// When zones get deleted on tracking end, the remaining distance to move reserved zones
// is limited to the windows up to the absolute window positions and the trackinglength backwards.
// Therefore from all windows of a TrackingLength - Startwindow is the distance 
// to be removed from the allowed shifting distance.
StartTrackingPosition := M_GetTrackingPosition((mStartWindowIndex-1)*WindowSize);
WindowsFromBegin := UDINT_TO_UINT(StartTrackingPosition / WindowSize);
WindowsTrackingLength := UDINT_TO_UINT((TrackingLength + TrackingAddition) / WindowSize);

IF WindowsFromBegin MOD WindowSize > 0 THEN
	WindowsFromBegin := WindowsFromBegin + 1;
END_IF

IF WindowsTrackingLength MOD WindowSize > 0 THEN
	WindowsTrackingLength := WindowsTrackingLength + 1;
END_IF

IF DeleteZoneTrackingEnd THEN	
	RemainingWindowLength := UINT_TO_INT(WindowsFromBegin) + UINT_TO_INT(WindowsTrackingLength) - UINT_TO_INT(ResWindowsToShift) - 1;
ELSE
	RemainingWindowLength := UINT_TO_INT(MaxWindowIndex) - UINT_TO_INT(ResWindowsToShift) - 1;
END_IF
	
FOR mIdx := 1 TO WindowTracking.MAX_NUMBER_OF_WINDOWS DO
	// Correct window border overflow
	IF mWindowIndex > MaxWindowIndex THEN
		mWindowIndex := mWindowIndex - MaxWindowIndex;
	END_IF
	
	IF mNextTargetWindow > MaxWindowIndex THEN
		mNextTargetWindow := mNextTargetWindow - MaxWindowIndex;
	END_IF
	
	// Relocation is done, if all zones in the shifting distance
	// and all interfering zones are relocated properly
	IF mIdx > ResWindowsToShift THEN
		M_IsShiftable := TRUE;
		EXIT;

	// If window is part of zone, try to schedule relocation
	ELSIF WindowTable[mWindowIndex].ZoneIndex > 0 THEN
		// Calculate Window Length of Zone which should be relocated
		mZoneIndexReloc := WindowTable[mWindowIndex].ZoneIndex;
		
		IF ZoneTable[mZoneIndexReloc].TU_Present THEN
			// Skip all occupied zones, because they are not allowed for re-allocation, otherwise fail
			IF mExcludeTUs THEN
				mWindowIndex := mWindowIndex + 1;
				RemainingWindowLength := RemainingWindowLength - 1;
				CONTINUE;
			ELSE
				M_IsShiftable := FALSE;
				EXIT;
			END_IF
		END_IF

		IF ZoneTable[mZoneIndexReloc].ZoneEndWindowIndex > ZoneTable[mZoneIndexReloc].ZoneStartWindowIndex THEN
			mWindowLength := ZoneTable[mZoneIndexReloc].ZoneEndWindowIndex - ZoneTable[mZoneIndexReloc].ZoneStartWindowIndex + 1;
		ELSE
			mWindowLength := ZoneTable[mZoneIndexReloc].ZoneEndWindowIndex + MaxWindowIndex  - ZoneTable[mZoneIndexReloc].ZoneStartWindowIndex + 1;
		END_IF

		// Check if reallocation would overwrite start point
		IF RemainingWindowLength - UINT_TO_INT(mWindowLength) > 0 THEN
			RelocScheduled := mfbRelocator.M_ScheduleRelocation(
									mZoneIndex				:= mZoneIndexReloc, 
									mTargetWindow			:= mNextTargetWindow, 
									mMaxWindowIndex			:= MaxWindowIndex, 
									mrWindowTable			:= WindowTable, 
									mrZoneTable				:= ZoneTable, 
									mBlockingZoneIndex		=> BlockingZoneIndex, 
									mBlockingEndWindowIndex => BlockingEndWindowIndex,
									mErrorId				=> ErrorId);
									
			// If relocation could be scheduled properly
			// set next window to the window after the relocated zone
			IF RelocScheduled THEN
				mNextTargetWindow := mNextTargetWindow + mWindowLength;
				
				// Adjust index of next window to check if relocation was successful
				mWindowIndex := mWindowIndex + mWindowLength;
				
				// Each found zone on the shifting distance requires one additional shift iteration
				// Because the location where it was moved to, may contains as well a zone which needs to be shifted
				ResWindowsToShift := ResWindowsToShift + 1;
				
				// Ensure that reallocation does not overwrite start point
				RemainingWindowLength := RemainingWindowLength - UINT_TO_INT(mWindowLength);
			ELSE
				// Relocation was not possible because of a Zone which is not allowed
				// to be shifted, try again with window after the blocking zone
				IF BlockingZoneIndex > 0 THEN
					// Each found zone on the shifting distance requires one additional shift iteration
					ResWindowsToShift := ResWindowsToShift + 1;
					
					// Calc length of blocking zone
					IF ZoneTable[BlockingZoneIndex].ZoneEndWindowIndex >= ZoneTable[BlockingZoneIndex].ZoneStartWindowIndex THEN
						mWindowLengthBlocking := ZoneTable[BlockingZoneIndex].ZoneEndWindowIndex - ZoneTable[BlockingZoneIndex].ZoneStartWindowIndex;
					ELSE
						mWindowLengthBlocking := ZoneTable[BlockingZoneIndex].ZoneEndWindowIndex + MaxWindowIndex - ZoneTable[BlockingZoneIndex].ZoneStartWindowIndex;
					END_IF
					
					mNextTargetWindow := BlockingEndWindowIndex + 1;
					
					RemainingWindowLength := RemainingWindowLength - UINT_TO_INT(mWindowLengthBlocking);
				END_IF
			END_IF
		ELSE
			// The found zone could not be placed on the tracking because there is no space left.
			// Mark overrun and leave
			mZoneOverrun := TRUE;
			mZoneOverrunWindowIndex := mWindowIndex;
			M_IsShiftable := mAllowOverrun;
			EXIT;
		END_IF
	ELSE
		mWindowIndex := mWindowIndex + 1;
		RemainingWindowLength := RemainingWindowLength - 1;
	END_IF
END_FOR
END_METHOD

/// Checks if a TU or a part of it, is found in a certain range.
METHOD M_IsTU_InRange : BOOL; // Returns true if present, otherwise false
VAR_INPUT
	mZoneIndex				: UINT; // Tracking zone index
	mAbsoluteStartRange		: UDINT; // Start range position on the tracking [mm]
	mAbsoluteEndRange		: UDINT; // End range position on the tracking [mm]
END_VAR
VAR
	mStartWindowIndex		: UINT; // Window index at start position
	mEndWindowIndex			: UINT; // Window index at end position
	mTrackingRangeEnd		: UDINT; // Tracking range position end
	mTrackingRangeStart		: UDINT; // Tracking range position start
	mTrackingTU_End			: UDINT; // Tracking range position end
	mTrackingTU_Start		: UDINT; // Tracking range position start
END_VAR
M_IsTU_InRange := FALSE;

// Check inputs
IF mZoneIndex = 0 THEN
	RETURN;
END_IF

IF NOT ZoneTable[mZoneIndex].TU_Present THEN
	RETURN;
END_IF

// Get window index of window start position
mStartWindowIndex := M_GetWindowIndex(mAbsoluteStartRange);
// Get window index of window end position
mEndWindowIndex := M_GetWindowIndex(mAbsoluteEndRange);

// Remark:
// Absolute view is unequal to tracking view
// ABS:  500mm 505mm .....1000mm
//   AbsStartpos		AbsEndPos
//       |                  |
//    TrackingEnd       TrackingStart
//
//  --------------------------------------      FlowDirection ->
// Win:  54  53  52 ....  43 42 ...
// Window index of end is normally lower than start (except overflow)     

// Ensure both window index are in a valid range
IF mStartWindowIndex > 0 AND mStartWindowIndex <= WindowTracking.MAX_NUMBER_OF_WINDOWS AND
   mEndWindowIndex > 0 AND mEndWindowIndex <= WindowTracking.MAX_NUMBER_OF_WINDOWS THEN
	
	// Ensure that Zone consists of start and end tu window index
	IF ZoneTable[mZoneIndex].TU_StartWindowIndex > 0 AND
	   ZoneTable[mZoneIndex].TU_EndWindowIndex > 0 THEN
	   
		//    TrackingEnd       TrackingStart
		//         |-----------------|
		//  --------------------------------------      FlowDirection ->
	   	mTrackingTU_End := WindowTable[ZoneTable[mZoneIndex].TU_EndWindowIndex].TU_RearEdgePosition;
	   	mTrackingTU_Start :=  WindowTable[ZoneTable[mZoneIndex].TU_StartWindowIndex].TU_FrontEdgePosition;
	   
		//    TrackingRangeEnd  TrackingRangeStart
		//      |----------------------|
		//  --------------------------------------      FlowDirection ->
		mTrackingRangeEnd := M_GetTrackingPosition(mAbsoluteStartRange);
   		mTrackingRangeStart := M_GetTrackingPosition(mAbsoluteEndRange);
	   
		// When range does not consists of the overflow point
		IF mTrackingRangeEnd >= mTrackingRangeStart THEN 
			// Check if TU End edge is between range
			IF mTrackingTU_End >= mTrackingRangeStart AND
               mTrackingTU_End <= mTrackingRangeEnd THEN
				M_IsTU_InRange := TRUE;
				RETURN;
				
			// Check if TU start edge is between range
			ELSIF mTrackingTU_Start >= mTrackingRangeStart AND
                  mTrackingTU_Start <= mTrackingRangeEnd THEN
				M_IsTU_InRange := TRUE;
				RETURN;
				
			// Check if TU is overlapping full range
			ELSIF mTrackingTU_End >= mTrackingRangeEnd AND
                  mTrackingTU_Start <= mTrackingRangeStart THEN
				M_IsTU_InRange := TRUE;
				RETURN; 
			END_IF
		// If range is overlapping overflow point
		ELSE
			// Check if TU End edge is between range
			IF mTrackingTU_End >= mTrackingRangeStart OR  
               mTrackingTU_End <= mTrackingRangeEnd THEN
				M_IsTU_InRange := TRUE;
				RETURN;
				
			// Check if TU start edge is between range
			ELSIF mTrackingTU_Start >= mTrackingRangeStart OR  
               mTrackingTU_Start <= mTrackingRangeEnd THEN
				M_IsTU_InRange := TRUE;
				RETURN;
				
			// Check if TU is overlapping full range
			ELSIF mTrackingTU_End >= mTrackingRangeEnd AND
                  mTrackingTU_Start <= mTrackingRangeStart THEN
				M_IsTU_InRange := TRUE;
				RETURN; 
			END_IF
		END_IF
	END_IF
END_IF
END_METHOD

/// Returns if a physical TU is present at mAbsolutePosition
METHOD M_IsTU_Present : BOOL; // Returns true if present, otherwise false
VAR_INPUT
	mAbsolutePosition		: UDINT; // Absolute position on tracking length
END_VAR
VAR
	mWindowIndex			: UINT; // Window index at absolute position
	mTrackingPosition		: UDINT; // Current position on tracking
END_VAR
M_IsTU_Present := FALSE;

// Get window index of position
mWindowIndex := M_GetWindowIndex(mAbsolutePosition);

IF mWindowIndex > 0 AND mWindowIndex <= WindowTracking.MAX_NUMBER_OF_WINDOWS THEN
	// Get position on tracking
	mTrackingPosition := M_GetTrackingPosition(mAbsolutePosition);

	// Get TU state
	CASE WindowTable[mWindowIndex].State OF
		E_WindowTrackingWindowState.IDLE:
			M_IsTU_Present := FALSE;
			
		E_WindowTrackingWindowState.FRONT_EDGE:
			IF WindowTable[mWindowIndex].TU_FrontEdgePosition <= mTrackingPosition THEN
				M_IsTU_Present := TRUE;
			ELSE
				M_IsTU_Present := FALSE;
			END_IF
		
		E_WindowTrackingWindowState.REAR_EDGE:
			IF WindowTable[mWindowIndex].TU_RearEdgePosition > mTrackingPosition THEN
				M_IsTU_Present := TRUE;
			ELSE
				M_IsTU_Present := FALSE;
			END_IF
		
		E_WindowTrackingWindowState.OCCUPIED:
			M_IsTU_Present := TRUE;
	END_CASE
END_IF
END_METHOD

/// Checks if a zone or a part of it,  is found in a certain range.
METHOD M_IsZoneInRange : BOOL; // Returns true if zone is in range, otherwise false
VAR_INPUT
	mZoneIndex				: UINT; // Tracking zone index
	mAbsoluteStartRange		: UDINT; // Start range position on the tracking [mm]
	mAbsoluteEndRange		: UDINT; // End range position on the tracking [mm]
END_VAR
VAR
	mStartWindowIndex		: UINT; // Window index at start position
	mEndWindowIndex			: UINT; // Window index at end position
	mTrackingRangeEnd		: UDINT; // Tracking range position end
	mTrackingRangeStart		: UDINT; // Tracking range position start
	mTrackingZoneEnd		: UDINT; // Tracking range position zone end
	mTrackingZoneStart		: UDINT; // Tracking range position zone start
END_VAR
M_IsZoneInRange := FALSE;

// Check inputs
IF mZoneIndex = 0 THEN
	RETURN;
END_IF

// Get window index of window start position
mStartWindowIndex := M_GetWindowIndex(mAbsoluteStartRange);
// Get window index of window end position
mEndWindowIndex := M_GetWindowIndex(mAbsoluteEndRange);

// Remark:
// Absolute view is unequal to tracking view
// ABS:  500mm 505mm .....1000mm
//    Startpos			 EndPos
//       |                  |
//  --------------------------------------      FlowDirection ->
// Win:  54  53  52 ....  43 42 ...
// Window index of end is normally lower than start (except overflow)     

// Ensure both window index are in a valid range
IF mStartWindowIndex > 0 AND mStartWindowIndex <= WindowTracking.MAX_NUMBER_OF_WINDOWS AND
   mEndWindowIndex > 0 AND mEndWindowIndex <= WindowTracking.MAX_NUMBER_OF_WINDOWS THEN

	// Ensure that Zone consists of start and end tu window index
	IF ZoneTable[mZoneIndex].TU_StartWindowIndex > 0 AND
	   ZoneTable[mZoneIndex].TU_EndWindowIndex > 0 THEN

		//    TrackingEnd       TrackingStart
		//         |-----------------|
		//  --------------------------------------      FlowDirection ->
	   	mTrackingZoneEnd := ZoneTable[mZoneIndex].ZoneEndPosition;
	   	mTrackingZoneStart := ZoneTable[mZoneIndex].ZoneStartPosition;

		//    TrackingRangeEnd  TrackingRangeStart
		//      |----------------------|
		//  --------------------------------------      FlowDirection ->
		mTrackingRangeEnd := M_GetTrackingPosition(mAbsoluteStartRange);
   		mTrackingRangeStart := M_GetTrackingPosition(mAbsoluteEndRange);

		// When range does not consists of the overflow point
		IF mTrackingRangeEnd >= mTrackingRangeStart THEN 
			// Check if TU End edge is between range
			IF mTrackingZoneEnd >= mTrackingRangeStart AND
               mTrackingZoneEnd <= mTrackingRangeEnd THEN
				M_IsZoneInRange := TRUE;
				RETURN;
				
			// Check if TU start edge is between range
			ELSIF mTrackingZoneStart >= mTrackingRangeStart AND
                  mTrackingZoneStart <= mTrackingRangeEnd THEN
				M_IsZoneInRange := TRUE;
				RETURN;
				
			// Check if TU is overlapping full range
			ELSIF mTrackingZoneEnd >= mTrackingRangeEnd AND
                  mTrackingZoneStart <= mTrackingRangeStart THEN
				M_IsZoneInRange := TRUE;
				RETURN; 
			END_IF
			
		// If range is overlapping overflow point
		ELSE
			// Check if TU End edge is between range
			IF mTrackingZoneEnd >= mTrackingRangeStart OR  
               mTrackingZoneEnd <= mTrackingRangeEnd THEN
				M_IsZoneInRange := TRUE;
				RETURN;
				
			// Check if TU start edge is between range
			ELSIF mTrackingZoneStart >= mTrackingRangeStart OR  
                  mTrackingZoneStart <= mTrackingRangeEnd THEN
				M_IsZoneInRange := TRUE;
				RETURN;
				
			// Check if TU is overlapping full range
			ELSIF mTrackingZoneEnd >= mTrackingRangeEnd AND
                  mTrackingZoneStart <= mTrackingRangeStart THEN
				M_IsZoneInRange := TRUE;
				RETURN; 
			END_IF
		END_IF
	END_IF
END_IF
END_METHOD

/// Tries to free a certain area by the following options (Shift, Shorten, Delete)
METHOD PROTECTED M_MakeSpace : BOOL // Returns true if successfully
VAR_INPUT
	mStartWindowIndex		: UINT; // Start window index
	mWindowsToFree			: UINT; // Windows to free up (e.g. 1 only clears start window index)
	mAllowZoneDelete		: BOOL; // Allows to delete zones if they could not be modified or reloacted
END_VAR
VAR_INST
	MinFreeWindowIndex		: UINT; // Minimum window index until space has to be free 
	ShiftZonesOk			: BOOL; // Shift was executed
END_VAR
VAR
	mIdx					: UINT; // Iteration
	mWindowIndex			: UINT; // Temp window index
	mZoneIndex				: UINT; // Zone index
	mTU_StartInArea			: BOOL; // TU start found in area
	mTU_EndInArea			: BOOL; // TU end found in area
END_VAR
// Initialize
M_MakeSpace := FALSE;

// Validate inputs
IF mStartWindowIndex = 0 OR
   mStartWindowIndex > WindowTracking.MAX_NUMBER_OF_WINDOWS OR
   mWindowsToFree = 0 OR
   mWindowsToFree > WindowTracking.MAX_NUMBER_OF_WINDOWS OR
   WindowSize = 0 THEN
	RETURN;
END_IF

// Initialize for-loop values
mWindowIndex := mStartWindowIndex;

// Calculate minimum window index which has to be free 
// Example: Startwindow 49, windows to be free 4 (49, 50, 51, 52)
//                  |-------------->
// Window     53 | 52 | 51 | 50 | 49
MinFreeWindowIndex := mStartWindowIndex + mWindowsToFree - 1;
	
// Correct window border overflow
IF MinFreeWindowIndex > MaxWindowIndex THEN
	MinFreeWindowIndex := MinFreeWindowIndex - MaxWindowIndex;
END_IF

// Check for any occupied zone in the area to be free and test if it spossible to shorten or delete it
FOR mIdx := 1 TO mWindowsToFree DO	
	IF WindowTable[mWindowIndex].ZoneIndex > 0 THEN
		mZoneIndex := WindowTable[mWindowIndex].ZoneIndex;
	
		// Zone can be modified by one of the following options
		// - If Occupied -> Shorten
		// - Else Delete if allowed
		IF ZoneTable[mZoneIndex].TU_Present THEN
			// Shorten
			// Check if position of TU inside the zone is outside of the area to be free
			IF MinFreeWindowIndex >= mStartWindowIndex THEN
				mTU_StartInArea := ZoneTable[mZoneIndex].TU_StartWindowIndex >= mStartWindowIndex AND
				   				   ZoneTable[mZoneIndex].TU_StartWindowIndex <= MinFreeWindowIndex;
				
				mTU_EndInArea := ZoneTable[mZoneIndex].TU_EndWindowIndex >= mStartWindowIndex AND
				   				 ZoneTable[mZoneIndex].TU_EndWindowIndex <= MinFreeWindowIndex;
				
			// Otherwise overflow between
			ELSE
				mTU_StartInArea := ZoneTable[mZoneIndex].TU_StartWindowIndex <= MinFreeWindowIndex OR
				   				   ZoneTable[mZoneIndex].TU_StartWindowIndex >= mStartWindowIndex;
				
				mTU_EndInArea := ZoneTable[mZoneIndex].TU_EndWindowIndex <= MinFreeWindowIndex OR
				   				 ZoneTable[mZoneIndex].TU_EndWindowIndex >= mStartWindowIndex;
			END_IF
			
			// TU Start or End is in area to be free
			IF mTU_StartInArea OR mTU_EndInArea THEN
				// Shorten not possible, check if delete is an option
				IF mAllowZoneDelete THEN
					// Ok
					;
				ELSE
					// Abort, shorten does not help
					M_MakeSpace := FALSE;
					RETURN;
				END_IF
			ELSE
				// Shorten is possible
				;
			END_IF
		END_IF
	END_IF
	
	mWindowIndex := mWindowIndex + 1;
	
	IF mWindowIndex > MaxWindowIndex THEN
		mWindowIndex := mWindowIndex - MaxWindowIndex;
	END_IF
END_FOR

// All occupied zones can be handled, try to shift 
ShiftZonesOk := M_ShiftZone(
					mStartWindowIndex,
					mWindowsToFree,
					TRUE,
					TRUE);

IF ShiftZonesOk THEN
	// First shorten zones at borders
	IF WindowTable[mStartWindowIndex].ZoneIndex > 0 THEN
		// If it consists of a TU
		IF ZoneTable[WindowTable[mStartWindowIndex].ZoneIndex].TU_Present THEN
			M_ShortenZoneAtWindow(
				WindowTable[mStartWindowIndex].ZoneIndex,
				mStartWindowIndex);
		END_IF
	END_IF

	IF WindowTable[MinFreeWindowIndex].ZoneIndex > 0 THEN
		// If it consists of a TU
		IF ZoneTable[WindowTable[MinFreeWindowIndex].ZoneIndex].TU_Present THEN
			M_ShortenZoneAtWindow(
				WindowTable[MinFreeWindowIndex].ZoneIndex,
				MinFreeWindowIndex);
		END_IF
	END_IF

	// Initialize loop
	mWindowIndex := mStartWindowIndex;
	
	// Execute TU operations
	FOR mIdx := 1 TO mWindowsToFree DO
		IF WindowTable[mWindowIndex].ZoneIndex > 0 THEN
			M_DeleteZone(WindowTable[mWindowIndex].ZoneIndex);
		END_IF
		
		mWindowIndex := mWindowIndex + 1;
	
		IF mWindowIndex > MaxWindowIndex THEN
			mWindowIndex := mWindowIndex - MaxWindowIndex;
		END_IF
	END_FOR
	
	M_MakeSpace := TRUE;
END_IF

IF NOT M_MakeSpace THEN
	// Error
	fbDebugMsg.M_SendErrorMsg('M_MakeSpace - Make space requested, but could not successfully executed.');	
END_IF
END_METHOD

/// Tries to free a certain area by the following options (Shift, Shorten, Delete)
METHOD PROTECTED M_MakeSpaceByWindows : BOOL // Returns true if successfully
VAR_INPUT
	mAbsolutePosition		: UDINT; // Start position window index
	mWindowsToFree			: UINT; // Windows to free up (e.g. 1 only clears start window index)
	mAllowZoneDelete		: BOOL; // Allows to delete zones if they could not be modified or reloacted
END_VAR

VAR
	mPositionWindowIndex	: UINT; // Window of position
END_VAR
M_MakeSpaceByWindows := FALSE;

// Validate inputs
IF WindowSize = 0 OR
   mWindowsToFree <= 0 THEN
	RETURN;
END_IF

mPositionWindowIndex := M_GetWindowIndex(mAbsolutePosition);

M_MakeSpaceByWindows := M_MakeSpace(
							mStartWindowIndex	:= mPositionWindowIndex, 
							mWindowsToFree		:= mWindowsToFree, 
							mAllowZoneDelete	:= mAllowZoneDelete);
END_METHOD

/// Allocates windows for ongoing transfers onto the belt 
/// until transfer gets completed by M_AddTU_RearEdge
/// Remark: Zones found during that process are tried to be shifted, otherwise deleted
METHOD PROTECTED M_ManageOngoingTransfers
VAR
	mIdx 				: UINT; // Loop iterator
	mWindowIndex		: UINT; // Current window iterator
	mTransferZoneIndex 	: UINT; // Transfer zone index iterator
	mFreeOk				: BOOL; // Shift ok
END_VAR
// Handle ongoing transfers onto the tracking belt
FOR mIdx := 1 TO TRANSFER_TABLE_SIZE DO
	// Check if dataset is active
	IF OngoingTransferList[mIdx].Active THEN
		// Get window index
		mWindowIndex := M_GetWindowIndex(OngoingTransferList[mIdx].AbsoluteInsertPosition);
		// Check if window has changed since last time
		IF mWindowIndex <> OngoingTransferList[mIdx].LastWindowIndex THEN
			IF mWindowIndex > 0 AND mWindowIndex <= WindowTracking.MAX_NUMBER_OF_WINDOWS THEN
				mTransferZoneIndex := OngoingTransferList[mIdx].ZoneIndex;
			
				// When a window gets overwritten which is already part of another zone, try to shift
				IF WindowTable[mWindowIndex].ZoneIndex > 0 AND
				   WindowTable[mWindowIndex].ZoneIndex <> mTransferZoneIndex THEN
					// Shift reserved zones
					mFreeOk := M_MakeSpaceByWindows(OngoingTransferList[mIdx].AbsoluteInsertPosition, 1, TRUE);
					
					// If not possible to shift, try to delete
					IF mFreeOk THEN
						DebugMsg := CONCAT('M_ManageOngoingTransfers - Could not free space. Zone: ',UINT_TO_STRING(WindowTable[mWindowIndex].ZoneIndex));
						fbDebugMsg.M_SendInfoMsg(DebugMsg);
					END_IF
				END_IF
				
				// A zone index needs to be available
				IF mTransferZoneIndex > 0 THEN
					// Update zone as currently end of TU, even this is not the last window to ensure always valid zone configuration
					// Otherwise it is unclear how many windows are part of a zone.
					WindowTable[mWindowIndex].State := E_WindowTrackingWindowState.REAR_EDGE;
					WindowTable[mWindowIndex].TU_RearEdgePosition := mWindowIndex * WindowSize - 1;
					
					WindowTable[mWindowIndex].ZoneIndex := OngoingTransferList[mIdx].ZoneIndex;
					ZoneTable[mTransferZoneIndex].ZoneEndWindowIndex := mWindowIndex;
					ZoneTable[mTransferZoneIndex].TU_EndWindowIndex := mWindowIndex;
					ZoneTable[mTransferZoneIndex].ZoneEndPosition := mWindowIndex * WindowSize - 1;
					
					
					IF ZoneTable[mTransferZoneIndex].ZoneEndPosition >= ZoneTable[mTransferZoneIndex].ZoneStartPosition THEN
						ZoneTable[mTransferZoneIndex].ZoneLength := UDINT_TO_UINT(ZoneTable[mTransferZoneIndex].ZoneEndPosition 
																				   - ZoneTable[mTransferZoneIndex].ZoneStartPosition);
					ELSE
						ZoneTable[mTransferZoneIndex].ZoneLength := UDINT_TO_UINT(ZoneTable[mTransferZoneIndex].ZoneEndPosition 
																				  + TotalTrackingLength 
																				  - ZoneTable[mTransferZoneIndex].ZoneStartPosition);
					END_IF
					
					// When a last is available (Was last rear edge, update to occupied 
					IF OngoingTransferList[mIdx].LastWindowIndex > 0 THEN
						IF WindowTable[OngoingTransferList[mIdx].LastWindowIndex].State = E_WindowTrackingWindowState.REAR_EDGE THEN
							WindowTable[OngoingTransferList[mIdx].LastWindowIndex].State := E_WindowTrackingWindowState.OCCUPIED;
							WindowTable[OngoingTransferList[mIdx].LastWindowIndex].TU_RearEdgePosition := 0;
						END_IF
					END_IF
					
					// Update transfer list
					OngoingTransferList[mIdx].LastWindowIndex := mWindowIndex;
				ELSE
					// Error
					;
				END_IF
			END_IF
		END_IF	
	ELSE
		EXIT;
	END_IF
END_FOR
END_METHOD

/// Monitors if one of the registered zones reach PTL, so they can be deleted
METHOD PROTECTED M_MonitorZonesPTL
VAR
	mIdx 				: UINT; // Loop iterator
	mPosition			: UDINT; // Current zone end position
END_VAR
// Handle ongoing ptl on the tracking distance
FOR mIdx := 1 TO MAX_NUMBER_OF_ZONES DO
	// Check if dataset is active
	IF PTL_Zones[mIdx] > 0 THEN		
		mPosition := M_GetZoneEndPosition(PTL_Zones[mIdx]);
		
		// Zone which consists of a TU or which are not valid anymore
		// get deleted from list, so they are not monitored anymore
		IF NOT ZoneTable[PTL_Zones[mIdx]].Used OR
		   ZoneTable[PTL_Zones[mIdx]].TU_Present THEN
			M_RemoveZoneFromPTL(PTL_Zones[mIdx]);
			
		// When the absolute position of zone end is reached, delete zone
		ELSIF mPosition > ZoneTable[PTL_Zones[mIdx]].PositionToLive AND mPosition < ZoneTable[PTL_Zones[mIdx]].PositionToLive + TrackingLength THEN
			M_DeleteZone(PTL_Zones[mIdx]);
		END_IF
	ELSE
		EXIT;
	END_IF
END_FOR
END_METHOD

/// Moves all windows of a zone to another target window. (Possible edges are applied as before in the new window)
/// Remark: Possible zones at destination get shifted or deleted based on configuration if possible.
METHOD PROTECTED M_MoveZone : BOOL // Returns true if successfully moved, otherwise false (e.g. target consists of a non movable zone)
VAR_INPUT
	mZoneIndex				: UINT; // Zone index to move
	mTargetStartWindow 		: UINT; // Target start window index
	mEnableDeleteOfZones  	: BOOL; // Zones at target destination gets deleted if they can not be shifted or shortened
END_VAR

VAR
	mIdx 					: UINT; // Loop iterator
	mZoneWindowLength 		: UINT; // Length of zone to be moved
	mWindowIndex 			: UINT; // Iterator window index loop
	mBufferOk				: BOOL; // Command executed successfully
END_VAR

VAR_INST
	MovePossible			: BOOL;
	OldRelWindowPositionRE 	: UDINT; // Old relative window position rear edge
	OldRelWindowPositionFE 	: UDINT; // Old relative window position front edge
	OldRelZoneStartPosition : UDINT; // Old relative zone start position
	OldRelZoneEndPosition 	: UDINT; // Old relative zone end position
	fbWindowBuffer			: FB_MemRingBuffer; // Temporary storage of source windows
	WindowBuffer			: ARRAY[1..(MAX_MOVE_WINDOWS * SIZEOF(ST_WindowTrackingWindow))] OF BYTE; // Buffer storage
END_VAR
M_MoveZone := FALSE;

// Validate inputs
IF mZoneIndex <= 0 OR
   mZoneIndex > MAX_NUMBER_OF_ZONES OR
   mTargetStartWindow = 0 OR
   mTargetStartWindow > MaxWindowIndex  THEN
   RETURN;
END_IF

// Calculate length of zone to move [windows]
IF ZoneTable[mZoneIndex].ZoneEndWindowIndex > ZoneTable[mZoneIndex].ZoneStartWindowIndex THEN
	mZoneWindowLength := ZoneTable[mZoneIndex].ZoneEndWindowIndex - ZoneTable[mZoneIndex].ZoneStartWindowIndex + 1;
ELSE
	mZoneWindowLength := ZoneTable[mZoneIndex].ZoneEndWindowIndex + MaxWindowIndex - ZoneTable[mZoneIndex].ZoneStartWindowIndex + 1;
END_IF


mWindowIndex := mTargetStartWindow;
MovePossible := TRUE;

IF NOT mEnableDeleteOfZones THEN
	// Clear target
	FOR mIdx := 1 TO mZoneWindowLength DO
		// Check if target is free or already part of the same zone
		IF WindowTable[mWindowIndex].ZoneIndex > 0 AND
		   WindowTable[mWindowIndex].ZoneIndex <> mZoneIndex THEN
		   
			// Make sure destination is free
			MovePossible := M_MakeSpace(
								mWindowIndex,
								1,
								mEnableDeleteOfZones);
								
			IF NOT MovePossible THEN
				EXIT;
			END_IF
		END_IF
		
		mWindowIndex := mWindowIndex + 1;
			
		// Correct border overflow
		IF mWindowIndex > MaxWindowIndex THEN
			mWindowIndex := mWindowIndex - MaxWindowIndex;
		END_IF
	END_FOR
END_IF

// When target is clear to receive a zone
IF MovePossible THEN
	// Clear temporary window buffer
	fbWindowBuffer.A_Reset(
		pBuffer 	:= ADR(WindowBuffer), 
		cbBuffer 	:= SIZEOF(WindowBuffer));
	
	mWindowIndex := ZoneTable[mZoneIndex].ZoneStartWindowIndex; 
	
	// Source windows needs to be stored temporarly, because it is possible
	// that the new target is inside the existing window range.
	FOR mIdx := 1 TO mZoneWindowLength DO
		// Add existing window to buffer
		fbWindowBuffer.A_AddTail(
			pBuffer 	:= ADR(WindowBuffer), 
			cbBuffer 	:= SIZEOF(WindowBuffer), 
			pWrite 		:= ADR(WindowTable[mWindowIndex]), 
			cbWrite 	:= SIZEOF(WindowTable[mWindowIndex]));
			
		mBufferOk := fbWindowBuffer.bOk;
			
		// Clear source window
		M_ClearWindow(mWindowIndex);
		
		mWindowIndex := mWindowIndex + 1;
		
		// Correct border overflow
		IF mWindowIndex > MaxWindowIndex THEN
			mWindowIndex := mWindowIndex - MaxWindowIndex;
		END_IF
	END_FOR
	
	// Copy source window to destination and update zone information
	mWindowIndex := mTargetStartWindow;
	
	FOR mIdx := 1 TO mZoneWindowLength DO
		// Copy window by window to target
		fbWindowBuffer.A_RemoveHead(
			pBuffer 	:= ADR(WindowBuffer), 
			cbBuffer 	:= SIZEOF(WindowBuffer), 
			pRead 		:= ADR(WindowTable[mWindowIndex]), 
			cbRead 		:= SIZEOF(WindowTable[mWindowIndex]));
		
		mBufferOk := fbWindowBuffer.bOk;
		
		// Update begin and end of zone
		IF mIdx = 1 THEN
			ZoneTable[mZoneIndex].ZoneStartWindowIndex := mWindowIndex;
			
		ELSIF mIdx = mZoneWindowLength THEN
			ZoneTable[mZoneIndex].ZoneEndWindowIndex := mWindowIndex;
		END_IF
		
		// When the moved window is marked as Front edge, update zone and position based on new window
		IF WindowTable[mWindowIndex].State = E_WindowTrackingWindowState.FRONT_EDGE THEN
			ZoneTable[mZoneIndex].TU_StartWindowIndex := mWindowIndex;
			OldRelWindowPositionFE := WindowTable[mWindowIndex].TU_FrontEdgePosition MOD WindowSize;
			WindowTable[mWindowIndex].TU_FrontEdgePosition := OldRelWindowPositionFE + (mWindowIndex-1) * WindowSize;
			
		// When the moved window is marked as Rear edge, update zone and position based on new window	
		ELSIF WindowTable[mWindowIndex].State = E_WindowTrackingWindowState.REAR_EDGE THEN 
			ZoneTable[mZoneIndex].TU_EndWindowIndex := mWindowIndex;
			OldRelWindowPositionRE := WindowTable[mWindowIndex].TU_RearEdgePosition MOD WindowSize;
			WindowTable[mWindowIndex].TU_RearEdgePosition := OldRelWindowPositionRE + (mWindowIndex-1) * WindowSize;
		END_IF
		
		mWindowIndex := mWindowIndex + 1;
		
		// Correct border overflow
		IF mWindowIndex > MaxWindowIndex THEN
			mWindowIndex := mWindowIndex - MaxWindowIndex;
		END_IF
	END_FOR
	
	// Update zone start and end position to new windows
	OldRelZoneStartPosition := ZoneTable[mZoneIndex].ZoneStartPosition MOD WindowSize;
	OldRelZoneEndPosition := ZoneTable[mZoneIndex].ZoneEndPosition MOD WindowSize;
	
	ZoneTable[mZoneIndex].ZoneStartPosition := OldRelZoneStartPosition + (ZoneTable[mZoneIndex].ZoneStartWindowIndex-1) * WindowSize;
	ZoneTable[mZoneIndex].ZoneEndPosition := OldRelZoneEndPosition + (ZoneTable[mZoneIndex].ZoneEndWindowIndex-1) * WindowSize;
	
	// Inform listener
	IF iEventListener <> 0 THEN
		iEventListener.M_TrackingZoneMovedEvent(
			mTrackingZoneIndex 	:= mZoneIndex,
			mTrackingZoneData 	:= ZoneTable[mZoneIndex]);
	END_IF
	
	M_MoveZone := TRUE;
END_IF
END_METHOD

/// Moves all windows of a zone to another target window aligned on front edge.
/// Remark: Possible zones at destination get shifted or deleted based on configuration.
/// Remark: If a physical TU can be found at Target, move not possible
METHOD PROTECTED M_MoveZoneFE : BOOL // Returns true if successful moved, otherwise false 
VAR_INPUT
	mZoneIndex					: UINT; // Zone index to move
	mAbsoluteTargetPosition		: UDINT; // Absolute target position [mm]
	mDeleteTargetZones  		: BOOL; // Zones at target destination gets deleted, otherwise shifted
END_VAR

VAR
	mMoveOk						: BOOL; // Move to new window location was successful
	mFrontEdgeAdjusted			: BOOL; // Front edge successfull adjusted
END_VAR

VAR_INST
	WindowNumberFE 				: UINT; // Number of front edge window in zone
	TargetWindowIndex			: UINT; // Target window index
	TargetMoveWindowIndex		: UINT; // Target move window index
	ZoneWindowLength 			: UINT; // Length of zone to be moved
	EdgeWindowIndex				: UINT; // Edge window index of zone
	NewTrackingPosition			: UDINT; // New required tracking position
	OldZoneStartWindowIndex 	: UINT; // Old zone start window index (Rollback)
END_VAR
M_MoveZoneFE := FALSE;

// Validate inputs
IF mZoneIndex <= 0 OR
   mZoneIndex > MAX_NUMBER_OF_ZONES OR
   WindowSize = 0 THEN
   RETURN;
END_IF

// Get window index of target position
TargetWindowIndex := M_GetWindowIndex(mAbsoluteTargetPosition);
   
// Ensure window is valid and physically occupied
IF ZoneTable[mZoneIndex].TU_Present AND
   TargetWindowIndex > 0 AND TargetWindowIndex <= WindowTracking.MAX_NUMBER_OF_WINDOWS THEN
   
	// Calculate length of zone in windows
	IF ZoneTable[mZoneIndex].ZoneEndWindowIndex > ZoneTable[mZoneIndex].ZoneStartWindowIndex THEN
		ZoneWindowLength := ZoneTable[mZoneIndex].ZoneEndWindowIndex - ZoneTable[mZoneIndex].ZoneStartWindowIndex + 1;
	ELSE
		ZoneWindowLength := ZoneTable[mZoneIndex].ZoneEndWindowIndex + MaxWindowIndex  - ZoneTable[mZoneIndex].ZoneStartWindowIndex + 1;
	END_IF
	
	// Store front edge and position of it in zone
	EdgeWindowIndex := ZoneTable[mZoneIndex].TU_StartWindowIndex;
	
	IF EdgeWindowIndex >= ZoneTable[mZoneIndex].ZoneStartWindowIndex THEN
		WindowNumberFE := EdgeWindowIndex - ZoneTable[mZoneIndex].ZoneStartWindowIndex + 1;
	ELSE
		WindowNumberFE := EdgeWindowIndex + MaxWindowIndex - ZoneTable[mZoneIndex].ZoneStartWindowIndex + 1;
	END_IF
	
	// If an edge is available
	IF EdgeWindowIndex > 0 THEN
		IF TargetWindowIndex >= WindowNumberFE THEN
			TargetMoveWindowIndex := TargetWindowIndex - WindowNumberFE + 1;
		ELSE
			TargetMoveWindowIndex := TargetWindowIndex + MaxWindowIndex - WindowNumberFE + 1;
		END_IF
		
		// Store old window index for a possible rollback
		OldZoneStartWindowIndex := ZoneTable[mZoneIndex].ZoneStartWindowIndex;
		
		// Move zone to target
		mMoveOk := M_MoveZone(
						mZoneIndex 				:= mZoneIndex,
						mTargetStartWindow 		:= TargetMoveWindowIndex,
						mEnableDeleteOfZones 	:= FALSE);	
		
		// If zone could be moved to new location, 
		IF mMoveOk THEN
			NewTrackingPosition := M_GetTrackingPosition(mAbsoluteTargetPosition);
			
			// try to adapt edge position changes (Front edge and rear edge)
			mFrontEdgeAdjusted := M_AdjustFE(
									mWindowIndexFE 			:= TargetWindowIndex,
									mNewTrackingPosition 	:= NewTrackingPosition,
									mDeleteTargetZones 		:= mDeleteTargetZones);
		
			IF mFrontEdgeAdjusted THEN
				// Move successful
				M_MoveZoneFE := TRUE;
			
			// Edge could not be aligned -> Rollback and abort		
			ELSE
				mMoveOk := M_MoveZone(
							mZoneIndex 				:= mZoneIndex,
							mTargetStartWindow 		:= OldZoneStartWindowIndex,
							mEnableDeleteOfZones 	:= FALSE);
							
				IF NOT mMoveOk THEN
					// Error during rollback
					;
				END_IF
				
				M_MoveZoneFE := FALSE;
			END_IF		
											
		// Move was not possible -> Abort						
		ELSE
			M_MoveZoneFE := FALSE;
		END_IF	
		
	// Otherwise no front edge window found
	ELSE
		M_MoveZoneFE := FALSE;
	END_IF
// Zone not valid 
ELSE
	M_MoveZoneFE := FALSE;
END_IF
END_METHOD

/// Moves all windows of a zone to another target window aligned on rear edge.
/// Remark: Possible zones at destination get shifted or deleted based on configuration.
/// Remark: If a physical TU can be found at Target, move not possible
METHOD PROTECTED M_MoveZoneRE : BOOL // Returns true if successful moved, otherwise false 
VAR_INPUT
	mZoneIndex					: UINT; // Zone index to move
	mAbsoluteTargetPosition		: UDINT; // Absolute target position [mm]
	mDeleteTargetZones  		: BOOL; // Zones at target destination gets deleted, otherwise shifted
END_VAR

VAR
	mMoveOk						: BOOL; // Move to new window location was successful
	mRearEdgeAdjusted			: BOOL; // Rear edge adjusted successfully
END_VAR

VAR_INST
	TargetWindowIndex			: UINT; // Target window index
	TargetMoveWindowIndex		: UINT; // Target move window index
	ZoneWindowLength 			: UINT; // Length of zone to be moved
	EdgeWindowIndex				: UINT; // Edge window index of zone
	WindowNumberRE 				: UINT; // Number of window in zone
	NewTrackingPosition			: UDINT; // new required tracking position
	OldZoneStartWindowIndex 	: UINT; // Old zone start window index (Rollback)
END_VAR
M_MoveZoneRE := FALSE;

// Validate inputs
IF mZoneIndex <= 0 OR
   mZoneIndex > MAX_NUMBER_OF_ZONES OR
   WindowSize = 0 THEN
   RETURN;
END_IF

// Get window index of target position
TargetWindowIndex := M_GetWindowIndex(mAbsoluteTargetPosition);
   
// Ensure window is valid and physically occupied
IF ZoneTable[mZoneIndex].TU_Present AND
   TargetWindowIndex > 0 AND TargetWindowIndex <= WindowTracking.MAX_NUMBER_OF_WINDOWS THEN 
	// Calculate length of zone in windows
	IF ZoneTable[mZoneIndex].ZoneEndWindowIndex > ZoneTable[mZoneIndex].ZoneStartWindowIndex THEN
		ZoneWindowLength := ZoneTable[mZoneIndex].ZoneEndWindowIndex - ZoneTable[mZoneIndex].ZoneStartWindowIndex + 1;
	ELSE
		ZoneWindowLength := ZoneTable[mZoneIndex].ZoneEndWindowIndex + MaxWindowIndex  - ZoneTable[mZoneIndex].ZoneStartWindowIndex + 1;
	END_IF
	
	// Store rear edge and position of it in zone
	EdgeWindowIndex := ZoneTable[mZoneIndex].TU_EndWindowIndex;
	
	IF EdgeWindowIndex >= ZoneTable[mZoneIndex].ZoneEndWindowIndex THEN
		WindowNumberRE := EdgeWindowIndex - ZoneTable[mZoneIndex].ZoneEndWindowIndex + 1;
	ELSE
		WindowNumberRE := EdgeWindowIndex + MaxWindowIndex - ZoneTable[mZoneIndex].ZoneEndWindowIndex + 1;
	END_IF
	
	// If an rear edge was found
	IF EdgeWindowIndex > 0 THEN
		// Calculate offset to ensure that rear edge window is at target window after move operation
		IF TargetWindowIndex >= WindowNumberRE THEN
			TargetMoveWindowIndex := TargetWindowIndex - WindowNumberRE + 1;
		ELSE
			TargetMoveWindowIndex := TargetWindowIndex + MaxWindowIndex - WindowNumberRE + 1;
		END_IF
		
		// Store old window index for a possible rollback
		OldZoneStartWindowIndex := ZoneTable[mZoneIndex].ZoneStartWindowIndex;

		// Move zone to target 
		mMoveOk := M_MoveZone(
						mZoneIndex 				:= mZoneIndex,
						mTargetStartWindow 		:= TargetMoveWindowIndex,
						mEnableDeleteOfZones 	:= FALSE);	
		
		// If zone could be moved to new location, 
		IF mMoveOk THEN
			NewTrackingPosition := M_GetTrackingPosition(mAbsoluteTargetPosition);
			
			// try to adapt edge position changes (Front edge and rear edge)
			mRearEdgeAdjusted := M_AdjustRE(
									mWindowIndexRE 			:= TargetWindowIndex,
									mNewTrackingPosition 	:= NewTrackingPosition,
									mDeleteTargetZones 		:= mDeleteTargetZones);
		
			IF mRearEdgeAdjusted THEN
				// Move successful
				M_MoveZoneRE := TRUE;
			
			// Edge could not be aligned -> Rollback and abort		
			ELSE
				fbDebugMsg.M_SendErrorMsg('M_MoveZoneRE - Rear edge could no be adjusted.');	
			
				mMoveOk := M_MoveZone(
							mZoneIndex 				:= mZoneIndex,
							mTargetStartWindow 		:= OldZoneStartWindowIndex,
							mEnableDeleteOfZones 	:= FALSE);
							
				IF NOT mMoveOk THEN
					// Error during rollback
					fbDebugMsg.M_SendErrorMsg('M_MoveZoneRE - Rollback not possible.');	
				END_IF
				
				M_MoveZoneRE := FALSE;
			END_IF
												
		// Move was not possible -> Abort						
		ELSE
			M_MoveZoneRE := FALSE;
		END_IF
		
	// Otherwise no rear edge window found
	ELSE
		M_MoveZoneRE := FALSE;
	END_IF
// Zone not valid 
ELSE
	M_MoveZoneRE := FALSE;
END_IF
END_METHOD

/// Removes a zone from the ptl list and closes all gaps in list
METHOD PROTECTED M_RemoveZoneFromPTL : BOOL // Returns true if zone was found and deleted, otherwise false
VAR_INPUT
	mZoneIndex			: UINT; // Zone index to remove
END_VAR
VAR
	mIdx				: UINT; // Iterator
	mCloseGapsInList 	: BOOL; // Flag to close gaps
END_VAR
M_RemoveZoneFromPTL := FALSE;
mCloseGapsInList := FALSE;

// Clean entry in PTL list and close gaps in list
FOR mIdx := 1 TO MAX_NUMBER_OF_ZONES DO
	IF PTL_Zones[mIdx] <> 0  THEN	
		IF PTL_Zones[mIdx] = mZoneIndex THEN 
			// Clear entry and mark following to close gaps
			mCloseGapsInList := TRUE;
			PTL_Zones[mIdx] := 0;
			M_RemoveZoneFromPTL := TRUE;
			
		ELSIF mCloseGapsInList THEN
			// Close gaps
			PTL_Zones[mIdx-1] := PTL_Zones[mIdx];
			PTL_Zones[mIdx] := 0;
		END_IF
	ELSE
		// No entries available
		EXIT;
	END_IF
END_FOR
END_METHOD

/// Removes a zone from the transfer list and closes all gaps in list
METHOD PROTECTED M_RemoveZoneFromTransferList : BOOL // Returns true if zone was found and deleted, otherwise false
VAR_INPUT
	mZoneIndex			: UINT; // Zone index to remove
END_VAR
VAR
	mIdx				: UINT; // Iterator
	mCloseGapsInList 	: BOOL; // Flag to close gaps
END_VAR
M_RemoveZoneFromTransferList := FALSE;
mCloseGapsInList := FALSE;

// Clean entry in transfer list and close gaps in list
FOR mIdx := 1 TO TRANSFER_TABLE_SIZE DO
	IF OngoingTransferList[mIdx].Active THEN	
		IF OngoingTransferList[mIdx].ZoneIndex = mZoneIndex THEN 
			// Clear entry and mark following to close gaps
			mCloseGapsInList := TRUE;
			MEMSET(ADR(OngoingTransferList[mIdx]), 0, SIZEOF(OngoingTransferList[mIdx]));
			M_RemoveZoneFromTransferList := TRUE;
			
		ELSIF mCloseGapsInList THEN
			// Close gaps
			OngoingTransferList[mIdx-1] := OngoingTransferList[mIdx];
			MEMSET(ADR(OngoingTransferList[mIdx]), 0, SIZEOF(OngoingTransferList[mIdx]));
		END_IF
	ELSE
		// No entries available
		EXIT;
	END_IF
END_FOR
END_METHOD

/// Reserve a Zone on tracking
/// Remark: Target needs to be free
METHOD PROTECTED M_ReserveZone : UINT // Returns Zone index if successful, otherwise 0
VAR_INPUT
	mActionId						: INT; (* ID of action which requests zone - 
								     		(0 = Only reservation, but free to be used by other actions) *)
	mLength							: UINT; // Length of zone to allocate [mm]
	mStartWindowIndex 				: UINT; // Start window index
	mStartTrackingPosition			: UDINT; // Start tracking position of the zone in start window [mm]
	mInhibitShifting				: BOOL; // Mark zone as not shiftable
	miActionListener				: I_TrackingActionListener; // Action listener of the created zone
	mPositionToLive					: UDINT; // Absolute position until allocation gets deleted automatically if not used (0 = disabled)
END_VAR
VAR_INST
	ZoneIndex 						: UINT; // Allocated zone index
	MaxWindowPosition 				: UDINT; // Input check for required poition MAX
	MinWindowPosition 				: UDINT; // Input check for required poition MIN
END_VAR
VAR
	mIdx							: UINT; // Loop iterator
	mWindowIndex					: UINT; // Start window index
	mWindowLength					: UINT; // Zone length in windows
	mEndWindowIndex					: UINT; // End window index
	mReservationAllowed 			: BOOL; // Reservation valid (e.g. free space available)
	mZoneEndPosition				: UDINT; // Zone end position 
	mRelWindowPositionZoneStart 	: UDINT; // Relative position of zone start in window
	mFullLength						: UINT; // Full length to be allocated
END_VAR
M_ReserveZone := 0;

// Validate inputs
IF mLength <= 0 OR
   WindowSize = 0 OR
   mStartWindowIndex <= 0 OR
   mStartWindowIndex > WindowTracking.MAX_NUMBER_OF_WINDOWS THEN
   RETURN;
END_IF

// Get max and min tracking position of front edge window
MaxWindowPosition := (mStartWindowIndex) * WindowSize;
MinWindowPosition := (mStartWindowIndex-1) * WindowSize;

// Ensure that new tracking position is in range of window
IF mStartTrackingPosition < MinWindowPosition OR 
   mStartTrackingPosition >= MaxWindowPosition THEN
   RETURN;
END_IF

// Calculate relative position in first zone window
mRelWindowPositionZoneStart := mStartTrackingPosition MOD WindowSize;

// The relative position in the first window is added to the length, 
// in order to get the amount of windows which are allocated for that TU finally
mFullLength := mLength + UDINT_TO_UINT(mRelWindowPositionZoneStart);

// Convert length into number of windows
mWindowLength := mFullLength / WindowSize;
// If not the full length could be mapped in windows
// add an additional window
IF (mFullLength MOD WindowSize) > 0 THEN
	mWindowLength := mWindowLength + 1;
END_IF

mWindowIndex := mStartWindowIndex;
mReservationAllowed := TRUE;

// Ensure reservation is possible
FOR mIdx := 1 TO mWindowLength DO
	// When zone is not empty or marked as flush, abort
	IF WindowTable[mWindowIndex].ZoneIndex > 0  OR
	   WindowTable[mWindowIndex].Flush THEN
	   // Cancel resevation
	   mReservationAllowed := FALSE;
	   M_ReserveZone := 0;
	   
	   	// Error
		fbDebugMsg.M_SendErrorMsg('M_ReserveZone - Reservation not possible, no available space.');	
	   	RETURN;
	END_IF
	
	mWindowIndex := mWindowIndex + 1;
 
	// Correct border overflow
	IF mWindowIndex > MaxWindowIndex THEN
		mWindowIndex := mWindowIndex - MaxWindowIndex;
	END_IF
END_FOR

// When reservation is possible to be executed
IF mReservationAllowed THEN
	// Get new Zone index
	ZoneIndex := M_InsertNewZoneIndex();
	
	IF ZoneIndex > 0 THEN
		mWindowIndex := mStartWindowIndex;
		
		// Loop through all windows and assigne new zone
		FOR mIdx := 1 TO mWindowLength DO
		   // Clear window
			MEMSET(ADR(WindowTable[mWindowIndex]),0,SIZEOF(WindowTable[mWindowIndex]));
			
			WindowTable[mWindowIndex].ZoneIndex := ZoneIndex;
			WindowTable[mWindowIndex].State := E_WindowTrackingWindowState.RESERVED;
							
			mWindowIndex := mWindowIndex + 1;
		 
			// Correct border overflow
			IF mWindowIndex > MaxWindowIndex THEN
				mWindowIndex := mWindowIndex - MaxWindowIndex;
			END_IF
		END_FOR
		
		mEndWindowIndex := mStartWindowIndex + mWindowLength - 1;
		
		// Correct border overflow
		IF mEndWindowIndex > MaxWindowIndex THEN
			mEndWindowIndex := mEndWindowIndex - MaxWindowIndex;
		END_IF
		
		mZoneEndPosition := mStartTrackingPosition + mLength;
		
		IF mZoneEndPosition > TotalTrackingLength THEN
			mZoneEndPosition := mZoneEndPosition - TotalTrackingLength;
		END_IF 
		
		ZoneTable[ZoneIndex].Used := TRUE;
		ZoneTable[ZoneIndex].ActionId := mActionId;
		ZoneTable[ZoneIndex].ZoneStartWindowIndex := mStartWindowIndex;
		ZoneTable[ZoneIndex].ZoneStartPosition := mStartTrackingPosition;
		ZoneTable[ZoneIndex].ZoneEndWindowIndex := mEndWindowIndex;
		ZoneTable[ZoneIndex].ZoneEndPosition := mZoneEndPosition;
		ZoneTable[ZoneIndex].ZoneLength := mLength;
		ZoneTable[ZoneIndex].InhibitShifting := mInhibitShifting;
		ZoneTable[ZoneIndex].iActionListener := miActionListener;
		ZoneTable[ZoneIndex].PositionToLive := mPositionToLive;

		IF mPositionToLive > 0 THEN
			M_AddZoneToPTL(ZoneIndex);
		END_IF
		
		// Inform listener
		IF iEventListener <> 0 THEN
			iEventListener.M_TrackingZoneAddedEvent(ZoneIndex,ZoneTable[ZoneIndex]);
		END_IF
		
		M_ReserveZone := ZoneIndex;
	ELSE
		// Error
		fbDebugMsg.M_SendErrorMsg('M_ReserveZone - Could not find free zone.');	
	END_IF
END_IF
END_METHOD

/// This function synchronize only a Front edge to a specific position and calculates the new TU length.
/// Remark: Zone begin gets adjusted to new front edge position. Spare windows in front of front edge get removed.
/// Remark: If at absolute position no zone is found, it searchs to the left for next front edge
/// until "mMaxFrontEdgeDeviation" to synchronize.
METHOD M_ResyncOnlyFE : UINT // Returns > 0 of the synchronized Zone index, otherwise 0 (e.g. No Zone, No occupied zone)
VAR_INPUT
	mAbsolutePosition		: UDINT; // Absolute position [mm]
	mMaxFrontEdgeDeviation 	: UDINT; (* When zone can not be found at "Absolute position",
										a search upwards is executed to a limit of MaxFrontEdgeDeviation [mm]*)
END_VAR
VAR_INST
	MaxTrackingPosition		: UDINT; // Max tracking distance to search for a zone
	NewPositionFE			: UDINT; // New front edge position in tracking
	NumberOfDeviationWindows: UINT; // Number of windows for maximal edge deviation 
	ZoneIndex				: UINT; // Zone index
	ZoneWindowLength 		: UINT; // Length of zone to be moved
	ExistingWindowIndexFE	: UINT; // Existing front edge window index
	ResyncPossible			: BOOL; // Resync is possible
	OldWindowFE				: ST_WindowTrackingWindow; // Stored old front edge window
	DistanceToTU_End		: DINT; // Distance to found TU End
	DistanceToTU_Start		: DINT; // Distance to found TU start
END_VAR
VAR
	mNewWindowIndexFE		: UINT; // Actual window index
	mWindowIndex			: UINT; // Window index iterator
	mIdx					: UINT; // Loop iterator
	mZoneFreeOk				: BOOL; // Shift possible
	mNewZoneWindowLength	: UINT; // Length of windows of aligned zone
END_VAR
M_ResyncOnlyFE := 0;
ZoneIndex := 0;
NumberOfDeviationWindows := 0;
mNewZoneWindowLength := 0;
ResyncPossible := TRUE;

// Validate values
IF WindowSize = 0 THEN
	RETURN;
END_IF

// Get window index at position
mNewWindowIndexFE := M_GetWindowIndex(mAbsolutePosition);

// Find related ZoneIndex
IF mNewWindowIndexFE > 0 AND mNewWindowIndexFE <= WindowTracking.MAX_NUMBER_OF_WINDOWS THEN
	// Ensure that target window is not already a rear edge window 
	// This is not permitted, minimum zone is two window
	IF WindowTable[mNewWindowIndexFE].State = E_WindowTrackingWindowState.REAR_EDGE THEN
		ZoneIndex := 0;
		
	// Search correlating zone
	// Check from target window to the left until MaxFrontedgeDeviation
	ELSE
		// Calculate max number of allowed front deviation windows
		NumberOfDeviationWindows := UDINT_TO_UINT(mMaxFrontEdgeDeviation / WindowSize);
		
		// Add an additional window if rest of division was unequal 0
		IF mMaxFrontEdgeDeviation MOD WindowSize > 0 THEN
			NumberOfDeviationWindows := NumberOfDeviationWindows + 1;
		END_IF
		
		// Get max tracking position for valid zone
		MaxTrackingPosition := M_GetTrackingPosition(mAbsolutePosition - mMaxFrontEdgeDeviation);

		// Search for adjacent zone
		mWindowIndex := mNewWindowIndexFE;
				
		// Check all additional windows plus begin
		FOR mIdx := 1 TO NumberOfDeviationWindows + 1 DO
			// Correct window border overflow
			IF mWindowIndex > MaxWindowIndex THEN
				mWindowIndex := mWindowIndex - MaxWindowIndex;
			END_IF
			
			// Search next zone
			IF WindowTable[mWindowIndex].ZoneIndex > 0 THEN
				DistanceToTU_End := M_GetDistanceToTU_End(mAbsolutePosition, WindowTable[mWindowIndex].ZoneIndex);
				DistanceToTU_Start := M_GetDistanceToTU_Start(mAbsolutePosition, WindowTable[mWindowIndex].ZoneIndex);
			
				// When a found zone is valid, check if edge is in valid range
				IF WindowTable[mWindowIndex].State = E_WindowTrackingWindowState.Front_EDGE THEN
					// Check if it's not last deviation window to check
					IF mIdx < NumberOfDeviationWindows + 1 THEN
						// Return found zone
						ZoneIndex := WindowTable[mWindowIndex].ZoneIndex;
					ELSE
						// Check position in window for max deviation
						IF WindowTable[mWindowIndex].TU_FrontEdgePosition <= MaxTrackingPosition THEN			
							// Return found zone
							ZoneIndex := WindowTable[mWindowIndex].ZoneIndex;
						END_IF
					END_IF
					EXIT;
					
				// Ensure TU end has not passed resync position and TU begin has reacher in minimum MaxDeviation pos
				// Remark: >0 = It is infront of resync position 
				ELSIF DistanceToTU_End > 0 AND
					  DistanceToTU_Start <= UDINT_TO_DINT(mMaxFrontEdgeDeviation) THEN
					// Return found zone
					ZoneIndex := WindowTable[mWindowIndex].ZoneIndex;
					EXIT;
				END_IF
			END_IF
			
			mWindowIndex := mWindowIndex + 1;
		END_FOR 
	END_IF
END_IF

// Ensure zone is valid (Consists of a TU, adaption of FE possible)
IF ZoneIndex > 0 THEN
	// Only possible if zone consists of a physical TU
	IF ZoneTable[ZoneIndex].TU_Present THEN
		// Ensure that no other zone is between new front edge and old rear edge
		mWindowIndex := mNewWindowIndexFE;
		ResyncPossible := TRUE;
		
		// Calculate new zone length in windows
		IF ZoneTable[ZoneIndex].ZoneEndWindowIndex > mNewWindowIndexFE THEN
			mNewZoneWindowLength := ZoneTable[ZoneIndex].ZoneEndWindowIndex - mNewWindowIndexFE + 1;
		ELSE
			mNewZoneWindowLength := ZoneTable[ZoneIndex].ZoneEndWindowIndex + MaxWindowIndex - mNewWindowIndexFE + 1;
		END_IF
	
		// Ensure resync has space
		FOR mIdx := 1 TO mNewZoneWindowLength DO	
			// If found window is empty or already part of the zone
			IF WindowTable[mWindowIndex].ZoneIndex = 0 OR
			   WindowTable[mWindowIndex].ZoneIndex = ZoneIndex THEN
			   // Window is valid
			   ;
			
			// Otherwise another zone is found, try to shift
			ELSE
				mZoneFreeOk := M_MakeSpace(
									mStartWindowIndex 	:= mWindowIndex, 
									mWindowsToFree 		:= 1,
									mAllowZoneDelete 	:= TRUE);
									
				IF NOT mZoneFreeOk THEN
					// Error, zone could not be shifted -> abort
					ResyncPossible := FALSE;
					EXIT;
				END_IF
			END_IF
			  
			mWindowIndex := mWindowIndex + 1;

			// Correct window border overflow
			IF mWindowIndex > MaxWindowIndex THEN
				mWindowIndex := mWindowIndex - MaxWindowIndex;
			END_IF
		END_FOR  
	END_IF
END_IF

// Process when a valid zone could be found
IF ZoneIndex > 0 AND ResyncPossible THEN
	// Calculate length of existing zone in windows
	IF ZoneTable[ZoneIndex].ZoneEndWindowIndex > ZoneTable[ZoneIndex].ZoneStartWindowIndex THEN
		ZoneWindowLength := ZoneTable[ZoneIndex].ZoneEndWindowIndex - ZoneTable[ZoneIndex].ZoneStartWindowIndex + 1;
	ELSE
		ZoneWindowLength := ZoneTable[ZoneIndex].ZoneEndWindowIndex + MaxWindowIndex  - ZoneTable[ZoneIndex].ZoneStartWindowIndex + 1;
	END_IF
	
	// Get existing front edge window
	ExistingWindowIndexFE := ZoneTable[ZoneIndex].TU_StartWindowIndex;
		
	// When front edge window could be found
	IF ExistingWindowIndexFE > 0 THEN
		// Store old window, because its possible to overwrite existing position
		OldWindowFE := WindowTable[ExistingWindowIndexFE];
		M_ClearWindow(ExistingWindowIndexFE);
		
		// Copy old window to new
		WindowTable[mNewWindowIndexFE] := OldWindowFE;
		
		NewPositionFE := M_GetTrackingPosition(mAbsolutePosition);
		
		// Adapt edge position and zone length
		WindowTable[mNewWindowIndexFE].TU_FrontEdgePosition := NewPositionFE;
		ZoneTable[ZoneIndex].ZoneStartWindowIndex := mNewWindowIndexFE;
		ZoneTable[ZoneIndex].TU_StartWindowIndex := mNewWindowIndexFE;
		ZoneTable[ZoneIndex].ZoneStartPosition := NewPositionFE;
		
		IF ZoneTable[ZoneIndex].ZoneEndPosition >= ZoneTable[ZoneIndex].ZoneStartPosition THEN
			ZoneTable[ZoneIndex].ZoneLength := UDINT_TO_UINT(ZoneTable[ZoneIndex].ZoneEndPosition - ZoneTable[ZoneIndex].ZoneStartPosition);
		ELSE
			ZoneTable[ZoneIndex].ZoneLength := UDINT_TO_UINT(ZoneTable[ZoneIndex].ZoneEndPosition + TotalTrackingLength - ZoneTable[ZoneIndex].ZoneStartPosition);
		END_IF

		// Clean all windows to the right of this zone
		mWindowIndex := mNewWindowIndexFE - 1;
		
		FOR mIdx := 1 TO MaxWindowIndex DO	
			// Correct window border overflow
			IF mWindowIndex <= 0 THEN
				mWindowIndex := mWindowIndex + MaxWindowIndex;
			END_IF
			
			// When window right of the front edge is part of the same zone, clean it
			IF WindowTable[mWindowIndex].ZoneIndex = ZoneIndex THEN
				M_ClearWindow(mWindowIndex);
				mWindowIndex := mWindowIndex -1;
			// Otherwise no other windows to clean
			ELSE
				EXIT;
			END_IF
		END_FOR  
			
		// Fill gap windows to the left
		mWindowIndex := mNewWindowIndexFE;
				
		FOR mIdx := 1 TO mNewZoneWindowLength DO	
			// Correct window border overflow
			IF mWindowIndex > MaxWindowIndex THEN
				mWindowIndex := mWindowIndex - MaxWindowIndex;
			END_IF
			
			// Assign ZoneIndex to all windows
			WindowTable[mWindowIndex].ZoneIndex := ZoneIndex;
			
			// Overwrite all windows as occupied except begin and end
			IF WindowTable[mWindowIndex].State = E_WindowTrackingWindowState.FRONT_EDGE THEN
				;
			// Stop overwriting at rear edge window
            ELSIF WindowTable[mWindowIndex].State = E_WindowTrackingWindowState.REAR_EDGE THEN
				EXIT;
			ELSE
				// Assign ZoneIndex to all windows
				WindowTable[mWindowIndex].ZoneIndex := ZoneIndex;
				WindowTable[mWindowIndex].State := E_WindowTrackingWindowState.OCCUPIED;
			
				// Possible flush can be resettet, because of synchronization its valid again
				WindowTable[mWindowIndex].Flush := 0;
				WindowTable[mWindowIndex].TU_FrontEdgePosition := 0;
				WindowTable[mWindowIndex].TU_RearEdgePosition := 0;
			END_IF

			mWindowIndex := mWindowIndex + 1;
		END_FOR  
		
		M_ResyncOnlyFE := ZoneIndex;
	END_IF
END_IF
END_METHOD

/// This function synchronize only Rear edge to a specific position and calculates new TU length.
/// Remark: Zone end gets adjusted to new rear edge position. Spare windows after rear edge get removed.
/// Remark: If at absolute position no zone is found, it search to the right
/// until "mMaxFrontEdgeDeviation" to find one to synchronize.
METHOD M_ResyncOnlyRE : UINT // Returns > 0 of the synchronized Zone index, otherwise 0
VAR_INPUT
	mAbsolutePosition		: UDINT; // Absolute position [mm]
	mMaxRearEdgeDeviation 	: UDINT; (* When zone can not be found at "Absolute position",
										a search upwards is executed to a limit of MaxRearEdgeDeviation [mm]*)
END_VAR
VAR_INST
	MinTrackingPosition		: UDINT; // Min tracking distance to search for a zone
	NumberOfDeviationWindows: UINT; // Number of windows for maximal edge deviation 
	ZoneIndex				: UINT; // Zone index
	ResyncPossible			: BOOL; // Resync is possible
	ExistingWindowIndexRE	: UINT; // Existing rear edge window index
	ZoneWindowLength 		: UINT; // Length of zone to be moved
	OldWindowRE				: ST_WindowTrackingWindow; // Stored old rear edge window
	NewPositionRE			: UDINT; // New rear edge position in tracking
	DistanceToTU_End		: DINT; // Distance to found TU End
	DistanceToTU_Start		: DINT; // Distance to found TU start
END_VAR
VAR
	mZoneFreeOk				: BOOL; // Successfully
	mNewZoneWindowLength	: UINT; // Length of windows of aligned zone
	mNewWindowIndexRE		: UINT; // Actual window index
	mWindowIndex			: UINT; // Window index iterator
	mIdx					: UINT; // Loop iterator
END_VAR
M_ResyncOnlyRE := 0;
ZoneIndex := 0;
NumberOfDeviationWindows := 0;

// Validate values
IF WindowSize = 0 THEN
	RETURN;
END_IF

// Get window index at position
mNewWindowIndexRE := M_GetWindowIndex(mAbsolutePosition);

IF mNewWindowIndexRE > 0 AND mNewWindowIndexRE <= WindowTracking.MAX_NUMBER_OF_WINDOWS THEN
	// Ensure that target window is not already a front edge window 
	// This is not permitted, minimum zone is two window
	IF WindowTable[mNewWindowIndexRE].State = E_WindowTrackingWindowState.FRONT_EDGE THEN
		ZoneIndex := 0;
		
	// Search correlating zone
	// Check from target window to the right until MaxFrontedgeDeviation
	ELSE
		// Calculate max number of allowed rear edge deviation windows
		NumberOfDeviationWindows := UDINT_TO_UINT(mMaxRearEdgeDeviation / WindowSize);
		
		// Add an additional window if rest of division was unequal 0
		IF mMaxRearEdgeDeviation MOD WindowSize > 0 THEN
			NumberOfDeviationWindows := NumberOfDeviationWindows + 1;
		END_IF
		
		// Get min  tracking position for valid zone
		MinTrackingPosition := M_GetTrackingPosition(mAbsolutePosition + mMaxRearEdgeDeviation);

		// Search for a adjacent zone
		mWindowIndex := mNewWindowIndexRE;

		FOR mIdx := 1 TO NumberOfDeviationWindows + 1 DO	
			// Correct window border overflow
			IF mWindowIndex <= 0 THEN
				mWindowIndex := mWindowIndex + MaxWindowIndex;
			END_IF
			
			// Search next zone
			IF WindowTable[mWindowIndex].ZoneIndex > 0 THEN
				DistanceToTU_End := M_GetDistanceToTU_End(mAbsolutePosition, WindowTable[mWindowIndex].ZoneIndex);
				DistanceToTU_Start := M_GetDistanceToTU_Start(mAbsolutePosition, WindowTable[mWindowIndex].ZoneIndex);
			
				// When a rear edge was found check for valid range
				IF WindowTable[mWindowIndex].State = E_WindowTrackingWindowState.REAR_EDGE THEN
					// If it's not last deviation window to check
					IF mIdx < NumberOfDeviationWindows + 1 THEN
						// Return found zone
						ZoneIndex := WindowTable[mWindowIndex].ZoneIndex;
					ELSE
						// Check position in window for max deviation
						IF WindowTable[mWindowIndex].TU_RearEdgePosition >= MinTrackingPosition THEN			
							// Return found zone
							ZoneIndex := WindowTable[mWindowIndex].ZoneIndex;
						END_IF
					END_IF
					EXIT;
					
				// Ensure TU start has passed resync position and TU end has reached in minimum MaxDeviation pos
				// Remark: >0 = It is infront of resync position 
				ELSIF DistanceToTU_Start < 0 AND
                      DistanceToTU_End >= UDINT_TO_DINT(mMaxRearEdgeDeviation) THEN
				   	// Return found zone
					ZoneIndex := WindowTable[mWindowIndex].ZoneIndex;
					EXIT;
				END_IF
			END_IF
			
			mWindowIndex := mWindowIndex - 1;
		END_FOR 
	END_IF
END_IF

// Ensure zone is valid (Consists of a TU, adaption of RE possible)
IF ZoneIndex > 0 THEN
	// Only possible if zone consists of a physical TU
	IF ZoneTable[ZoneIndex].TU_Present THEN
		// Ensure that no other zone is between new rear edge and old front edge
		mWindowIndex := ZoneTable[ZoneIndex].ZoneStartWindowIndex;
		ResyncPossible := TRUE;
		
		// Calculate new zone length in windows
		IF mNewWindowIndexRE > ZoneTable[ZoneIndex].ZoneStartWindowIndex THEN
			mNewZoneWindowLength := mNewWindowIndexRE - ZoneTable[ZoneIndex].ZoneStartWindowIndex + 1;
		ELSE
			mNewZoneWindowLength := mNewWindowIndexRE  + MaxWindowIndex - ZoneTable[ZoneIndex].ZoneStartWindowIndex + 1;
		END_IF
	
		// Validate that sync is possible
		FOR mIdx := 1 TO mNewZoneWindowLength DO	
			// If found window is empty or already part of the zone
			IF WindowTable[mWindowIndex].ZoneIndex = 0 OR
			   WindowTable[mWindowIndex].ZoneIndex = ZoneIndex THEN
			   // Window is valid
			   ;
			
			// Otherwise another zone is found, try to shift
			ELSE
				mZoneFreeOk := M_MakeSpace(
									mStartWindowIndex 	:= mWindowIndex, 
									mWindowsToFree 		:= 1,
									mAllowZoneDelete 	:= TRUE);
									
				IF NOT mZoneFreeOk THEN
					// Error, zone could not be shifted -> abort
					ResyncPossible := FALSE;
					EXIT;
				END_IF
			END_IF
			  
			mWindowIndex := mWindowIndex + 1;

			// Correct window border overflow
			IF mWindowIndex > MaxWindowIndex THEN
				mWindowIndex := mWindowIndex - MaxWindowIndex;
			END_IF
		END_FOR  
	END_IF
END_IF

IF ZoneIndex > 0 AND ResyncPossible THEN
	// Calculate length of existing zone in windows
	IF ZoneTable[ZoneIndex].ZoneEndWindowIndex > ZoneTable[ZoneIndex].ZoneStartWindowIndex THEN
		ZoneWindowLength := ZoneTable[ZoneIndex].ZoneEndWindowIndex - ZoneTable[ZoneIndex].ZoneStartWindowIndex + 1;
	ELSE
		ZoneWindowLength := ZoneTable[ZoneIndex].ZoneEndWindowIndex + MaxWindowIndex  - ZoneTable[ZoneIndex].ZoneStartWindowIndex + 1;
	END_IF
	
	// Get existing rear edge window
	ExistingWindowIndexRE := ZoneTable[ZoneIndex].TU_EndWindowIndex;
	
	// When rear edge window could be found
	IF ExistingWindowIndexRE > 0 THEN
		// Store old window, because its possible to overwrite existing position
		OldWindowRE := WindowTable[ExistingWindowIndexRE];
		M_ClearWindow(ExistingWindowIndexRE);
		
		// Copy old window to new
		WindowTable[mNewWindowIndexRE] := OldWindowRE;
		
		NewPositionRE := M_GetTrackingPosition(mAbsolutePosition);
		
		// Adapt edge position and zone length
		WindowTable[mNewWindowIndexRE].TU_RearEdgePosition := NewPositionRE;
		ZoneTable[ZoneIndex].ZoneEndWindowIndex := mNewWindowIndexRE;
		ZoneTable[ZoneIndex].TU_EndWindowIndex := mNewWindowIndexRE;
		ZoneTable[ZoneIndex].ZoneEndPosition := NewPositionRE;
		
		IF ZoneTable[ZoneIndex].ZoneEndPosition >= ZoneTable[ZoneIndex].ZoneStartPosition THEN
			ZoneTable[ZoneIndex].ZoneLength := UDINT_TO_UINT(ZoneTable[ZoneIndex].ZoneEndPosition - ZoneTable[ZoneIndex].ZoneStartPosition);
		ELSE
			ZoneTable[ZoneIndex].ZoneLength := UDINT_TO_UINT(ZoneTable[ZoneIndex].ZoneEndPosition + TotalTrackingLength - ZoneTable[ZoneIndex].ZoneStartPosition);
		END_IF
		
		// Clean all windows to the left of this zone
		mWindowIndex := mNewWindowIndexRE + 1;
		
		FOR mIdx := 1 TO MaxWindowIndex DO	
			// Correct window border overflow
			IF mWindowIndex > MaxWindowIndex THEN
				mWindowIndex := mWindowIndex - MaxWindowIndex;
			END_IF
			
			// When window left of the rear edge is part of the same zone, clean it
			IF WindowTable[mWindowIndex].ZoneIndex = ZoneIndex THEN
				M_ClearWindow(mWindowIndex);
				mWindowIndex := mWindowIndex + 1;
			// Otherwise no other windows to clean
			ELSE
				EXIT;
			END_IF
		END_FOR  
			
		// Fill gap windows to the right
		mWindowIndex := mNewWindowIndexRE;
				
		FOR mIdx := 1 TO mNewZoneWindowLength DO	
			// Correct window border overflow
			IF mWindowIndex <= 0 THEN
				mWindowIndex := mWindowIndex + MaxWindowIndex;
			END_IF
			
			// Assign ZoneIndex to all windows
			WindowTable[mWindowIndex].ZoneIndex := ZoneIndex;
			
			// Overwrite all windows as occupied except begin and end
			IF WindowTable[mWindowIndex].State = E_WindowTrackingWindowState.REAR_EDGE THEN
				;
				
			// Stop overwriting at front edge window
            ELSIF WindowTable[mWindowIndex].State = E_WindowTrackingWindowState.FRONT_EDGE THEN
				EXIT;
				
			ELSE
				// Assign ZoneIndex to all windows
				WindowTable[mWindowIndex].ZoneIndex := ZoneIndex;
				WindowTable[mWindowIndex].State := E_WindowTrackingWindowState.OCCUPIED;
			
				// Possible flush can be reset, because of synchronization its valid again
				WindowTable[mWindowIndex].Flush := 0;
				WindowTable[mWindowIndex].TU_FrontEdgePosition := 0;
				WindowTable[mWindowIndex].TU_RearEdgePosition := 0;
			END_IF

			mWindowIndex := mWindowIndex - 1;
		END_FOR  
		
		M_ResyncOnlyRE := ZoneIndex;
	END_IF
END_IF
END_METHOD

/// This function synchronize whole TU aligned by Front edge to a specific position.
/// Rear edge is adjusted automatically to keep the length of TU.
/// Remark: If at absolute position no zone is found, it search to the left
/// until "mMaxFrontEdgeDeviation" to find one to synchronize.
METHOD M_ResyncTU_FE : UINT // Returns > 0 of the synchronized Zone index, otherwise 0
VAR_INPUT
	mAbsolutePosition		: UDINT; // Absolute position [mm]
	mMaxFrontEdgeDeviation 	: UDINT; (* When zone can not be found at "Absolute position",
										a search upwards is executed to a limit of MaxFrontEdgeDeviation [mm]*)
END_VAR
VAR_INST
	MaxTrackingPosition		: UDINT; // Max tracking distance to search for a zone
	NumberOfDeviationWindows: UINT; // Number of windows for maximal edge deviation 
	ZoneIndex				: UINT; // Zone index
END_VAR
VAR
	mZoneMoved 				: BOOL; // Zone moved successfully
	mSyncWindowIndex		: UINT; // Actual window index
	mWindowIndex			: UINT; // Window index iterator
	mIdx					: UINT; // Loop iterator
	DistanceToTU_End		: DINT; // Distance to found TU End
	DistanceToTU_Start		: DINT; // Distance to found TU start
END_VAR
M_ResyncTU_FE := 0;
ZoneIndex := 0;
NumberOfDeviationWindows := 0;

// Validate values
IF WindowSize = 0 THEN
	RETURN;
END_IF

// Get window index at position
mSyncWindowIndex := M_GetWindowIndex(mAbsolutePosition);

// Search correlating zone
// Check from target window to the left until MaxFrontedgeDeviation
IF mSyncWindowIndex > 0 AND mSyncWindowIndex <= WindowTracking.MAX_NUMBER_OF_WINDOWS THEN
	// Calculate max number of allowed front deviation windows
	NumberOfDeviationWindows := UDINT_TO_UINT(mMaxFrontEdgeDeviation / WindowSize);
	
	// Add an additional window if rest of division was unequal 0
	IF mMaxFrontEdgeDeviation MOD WindowSize > 0 THEN
		NumberOfDeviationWindows := NumberOfDeviationWindows + 1;
	END_IF
	
	// Get max tracking position for valid zone
	MaxTrackingPosition := M_GetTrackingPosition(mAbsolutePosition - mMaxFrontEdgeDeviation);

	// Search for adjacent zone
	mWindowIndex := mSyncWindowIndex;
			
	FOR mIdx := 1 TO NumberOfDeviationWindows + 1 DO	
		// Correct window border overflow
		IF mWindowIndex > MaxWindowIndex THEN
			mWindowIndex := mWindowIndex - MaxWindowIndex;
		END_IF
		
		// Search next zone
		IF WindowTable[mWindowIndex].ZoneIndex > 0 THEN
			DistanceToTU_End := M_GetDistanceToTU_End(mAbsolutePosition, WindowTable[mWindowIndex].ZoneIndex);
			DistanceToTU_Start := M_GetDistanceToTU_Start(mAbsolutePosition, WindowTable[mWindowIndex].ZoneIndex);
			
			// When a found zone is valid, check if edge is in valid range
			IF WindowTable[mWindowIndex].State = E_WindowTrackingWindowState.Front_EDGE THEN
				// Check if it's not last deviation window to check
				// Then it is anyway in the valid range
				IF mIdx < NumberOfDeviationWindows + 1 THEN
					// Return found zone
					ZoneIndex := WindowTable[mWindowIndex].ZoneIndex;
					
				// if it is the last window,
				// ensure the position inside the window is in the allowed border
				ELSE
					// Check position in window for max deviation
					IF WindowTable[mWindowIndex].TU_FrontEdgePosition <= MaxTrackingPosition THEN			
						// Return found zone
						ZoneIndex := WindowTable[mWindowIndex].ZoneIndex;
					END_IF
				END_IF
				EXIT;
				
			// Ensure TU end has not passed resync position and TU begin has reacher in minimum MaxDeviation pos
			// Remark: >0 = It is infront of resync position 
			ELSIF DistanceToTU_End > 0 AND
                  DistanceToTU_Start <= UDINT_TO_DINT(mMaxFrontEdgeDeviation) THEN
				// Return found zone
				ZoneIndex := WindowTable[mWindowIndex].ZoneIndex;
				EXIT;
			END_IF
		END_IF
		
		mWindowIndex := mWindowIndex + 1;
	END_FOR 
END_IF

// Process when a zone could be found
IF ZoneIndex > 0 THEN
	mZoneMoved := M_MoveZoneFE(
					mZoneIndex 				:= ZoneIndex,
					mAbsoluteTargetPosition := mAbsolutePosition,
					mDeleteTargetZones 		:= FALSE);
					
	IF mZoneMoved THEN
		M_ResyncTU_FE := ZoneIndex;
	ELSE
		M_ResyncTU_FE := 0;
	END_IF
END_IF
END_METHOD

/// This function synchronize whole TU aligned by Rear edge to a specific position.
/// Front edge is adjusted automatically to keep the length of TU.
/// Remark: If at absolute position no zone is found, it search to the right
/// until "mMaxFrontEdgeDeviation" to find one to synchronize.
METHOD M_ResyncTU_RE : UINT // Returns > 0 of the synchronized Zone index, otherwise 0
VAR_INPUT
	mAbsolutePosition		: UDINT; // Absolute position [mm]
	mMaxRearEdgeDeviation 	: UDINT; (* When zone can not be found at "Absolute position",
										a search upwards is executed to a limit of MaxRearEdgeDeviation [mm]*)
END_VAR
VAR_INST
	MinTrackingPosition		: UDINT; // Min tracking distance to search for a zone
	NumberOfDeviationWindows: UINT; // Number of windows for maximal edge deviation 
	ZoneIndex				: UINT; // Zone index
	DistanceToTU_End		: DINT; // Distance to found TU End
	DistanceToTU_Start		: DINT; // Distance to found TU start
END_VAR
VAR
	mZoneMoved 				: BOOL; // Zone moved successfully
	mSyncWindowIndex		: UINT; // Actual window index
	mWindowIndex			: UINT; // Window index iterator
	mIdx					: UINT; // Loop iterator
END_VAR
M_ResyncTU_RE := 0;
ZoneIndex := 0;
NumberOfDeviationWindows := 0;

// Validate values
IF WindowSize = 0 THEN
	RETURN;
END_IF

// Get window index at position
mSyncWindowIndex := M_GetWindowIndex(mAbsolutePosition);

IF mSyncWindowIndex > 0 AND mSyncWindowIndex <= WindowTracking.MAX_NUMBER_OF_WINDOWS THEN
	// Calculate max number of allowed rear edge deviation windows
	NumberOfDeviationWindows := UDINT_TO_UINT(mMaxRearEdgeDeviation / WindowSize);
	
	// Add an additional window if rest of division was unequal 0
	IF mMaxRearEdgeDeviation MOD WindowSize > 0 THEN
		NumberOfDeviationWindows := NumberOfDeviationWindows + 1;
	END_IF
	
	// Get min tracking position for valid zone
	MinTrackingPosition := M_GetTrackingPosition(mAbsolutePosition - mMaxRearEdgeDeviation);

	// Search for a adjacent zone to the right
	mWindowIndex := mSyncWindowIndex;
			
	FOR mIdx := 1 TO NumberOfDeviationWindows + 1 DO	
		// Correct window border overflow
		IF mWindowIndex <= 0 THEN
			mWindowIndex := mWindowIndex + MaxWindowIndex;
		END_IF
		
		// Search next zone
		IF WindowTable[mWindowIndex].ZoneIndex > 0 THEN
			DistanceToTU_End := M_GetDistanceToTU_End(mAbsolutePosition, WindowTable[mWindowIndex].ZoneIndex);
			DistanceToTU_Start := M_GetDistanceToTU_Start(mAbsolutePosition, WindowTable[mWindowIndex].ZoneIndex);
			
			// When a found zone is valid, check if edge is in valid range
			IF WindowTable[mWindowIndex].State = E_WindowTrackingWindowState.REAR_EDGE THEN
				// If it's not last deviation window to check
				IF mIdx < NumberOfDeviationWindows THEN
					// Return found zone
					ZoneIndex := WindowTable[mWindowIndex].ZoneIndex;
				ELSE
					// Check position in window for max deviation
					IF WindowTable[mWindowIndex].TU_RearEdgePosition >= MinTrackingPosition THEN
						// Return found zone
						ZoneIndex := WindowTable[mWindowIndex].ZoneIndex;
					END_IF
				END_IF
				EXIT;
				
			// Ensure TU start has passed resync position and TU end has reached in minimum MaxDeviation pos
			// Remark: >0 = It is infront of resync position 
			ELSIF DistanceToTU_Start < 0 AND
                  DistanceToTU_End >= UDINT_TO_DINT(mMaxRearEdgeDeviation) THEN
				 // Return found zone
				ZoneIndex := WindowTable[mWindowIndex].ZoneIndex;
				EXIT;
			END_IF
		END_IF
		
		mWindowIndex := mWindowIndex - 1;
	END_FOR 
END_IF

// Process when a zone could be found
IF ZoneIndex > 0 THEN
	mZoneMoved := M_MoveZoneRE(
					mZoneIndex 				:= ZoneIndex,
					mAbsoluteTargetPosition := mAbsolutePosition,
					mDeleteTargetZones 		:= FALSE);
					
	IF mZoneMoved THEN
		M_ResyncTU_RE := ZoneIndex;
	ELSE
		M_ResyncTU_RE := 0;
	END_IF
END_IF
END_METHOD

/// Shift zone at StartWindowIndex by WindowsToShift (If WindowsToShift includes more zones, they are shifted as well)
/// Remark: Only Zones without a TU Present and permition to shift, can be shifted. 
/// Remark: When a zone is found to shift, the whole zone is shifted
/// Remark: Zones which can not be reallocated (e.g. not enough space on tracking) get deleted. Owner of the Zone
/// will be notfied about that process.
METHOD PROTECTED M_ShiftZone : BOOL // Returns true if successfull shifted, otherwise false (e.g. not allowed to shift, wrong input)
VAR_INPUT
	mStartWindowIndex		: UINT; // Start window index
	mWindowsToShift			: UINT; // Windows to shift
	mExcludeTUs				: BOOL; // Exclude physical occupied zones
	mAllowOverrun			: BOOL; // Allow to throw out zones which cannot be place on the tracking anymore because of reallocations
END_VAR
VAR_INST
	ShiftingAllowed			: BOOL; // Target position is to be shifted
	RetrieveOk 				: BOOL; // Retrieve reallocation order successfully
	MoveOk 					: BOOL; // Move of zone executed successfully
	RelocEntry 				: ST_WindowTrackingReloc; // Reallocation order
	fbRelocator 			: FB_WindowRelocator; // Windows relocator
	ZoneOverrun				: BOOL;
	ZoneOverrunWindowIndex	: UINT;
END_VAR
VAR
	mIdx 					: DINT; // Loop iterator
	mNumberOfOverrunWindows : UINT;
	mEndOverrunWindowIndex	: UINT;
	mWindowIndex 			: UDINT; // Window index to loop trough tracking distance
END_VAR
M_ShiftZone := FALSE;

// Validate inputs
IF mStartWindowIndex = 0 OR
   mStartWindowIndex > WindowTracking.MAX_NUMBER_OF_WINDOWS OR
   mWindowsToShift = 0 OR
   mWindowsToShift > WindowTracking.MAX_NUMBER_OF_WINDOWS OR
   WindowSize = 0 THEN
	RETURN;
END_IF

// Inform listener
IF iEventListener <> 0 THEN
	iEventListener.M_TrackingShiftingInitiatedEvent(
		mAbsolutePosition 	:= M_GetAbsolutePosition(mStartWindowIndex - 1 * WindowSize),
		mDistance 			:= mWindowsToShift * WindowSize,
		mWindowIndex 		:= mStartWindowIndex,
		mWindowsToShift 	:= mWindowsToShift);
END_IF

fbRelocator.M_Reset();

ShiftingAllowed := M_IsShiftable(
						mStartWindowIndex,
						mWindowsToShift,
						mExcludeTUs,
						mAllowOverrun,
						mZoneOverrun => ZoneOverrun,
						mZoneOverrunWindowIndex => ZoneOverrunWindowIndex,
						mfbRelocator := fbRelocator);

IF ShiftingAllowed THEN
	// Clear overrun distance if allowed
	IF ZoneOverrun THEN
		IF mStartWindowIndex = 1 THEN
			mEndOverrunWindowIndex := MaxWindowIndex;
		ELSE	
			mEndOverrunWindowIndex := mStartWindowIndex - 1;
		END_IF
	
		IF mEndOverrunWindowIndex >= ZoneOverrunWindowIndex THEN
			mNumberOfOverrunWindows := mEndOverrunWindowIndex - ZoneOverrunWindowIndex;
		ELSE
			mNumberOfOverrunWindows := mEndOverrunWindowIndex + MaxWindowIndex - ZoneOverrunWindowIndex;
		END_IF
		
		mWindowIndex := ZoneOverrunWindowIndex;
		
		// Clear all zones which can not be relocated
		FOR mIdx := 1 TO mNumberOfOverrunWindows DO
			IF WindowTable[mWindowIndex].ZoneIndex > 0 THEN
				M_DeleteZone(WindowTable[mWindowIndex].ZoneIndex);
			END_IF
			
			mWindowIndex := mWindowIndex + 1;
			
			IF mWindowIndex > MaxWindowIndex THEN
				mWindowIndex := mWindowIndex - MaxWindowIndex;
			END_IF
		END_FOR
	END_IF

	// Do reallocation
	// Execute all scheduled reallocations
	FOR mIdx := 1 TO MAX_NUMBER_OF_ZONES DO
		
		RetrieveOk := fbRelocator.M_RetrieveLastEntry(
						mpData 		:= ADR(RelocEntry),
						mDataSize 	:= SIZEOF(RelocEntry));
						
		// Move all zones according all stored reallocation orders starting with the last added
		IF RetrieveOk THEN
			MoveOk := M_MoveZone(
						mZoneIndex 				:= RelocEntry.ZoneIndex,
						mTargetStartWindow 		:= RelocEntry.TargetWindow,
						mEnableDeleteOfZones 	:= TRUE);
						
			IF NOT MoveOk THEN
				// Error
				fbDebugMsg.M_SendErrorMsg('M_ShiftZone - Move was not possible.');	
			END_IF
		ELSE
			// No entries available anymore
			EXIT;
		END_IF
	END_FOR
	
	// Shifting executed
	M_ShiftZone := TRUE;
ELSE
	M_ShiftZone := FALSE;
END_IF

// Inform listener
IF iEventListener <> 0 THEN
	iEventListener.M_TrackingShiftingCompletedEvent(
		mAbsolutePosition 	:= M_GetAbsolutePosition(mStartWindowIndex - 1 * WindowSize),
		mDistance 			:= mWindowsToShift * WindowSize,
		mWindowIndex 		:= mStartWindowIndex,
		mWindowsToShift 	:= mWindowsToShift);
END_IF
END_METHOD

/// Shortens a zone by given value in up- or downstream direction
METHOD M_ShortenZone : BOOL// Returns TRUE if successful,
VAR_INPUT
	mZoneIndex 				: UINT; // Zone index to enlarge
	mReductionLength		: UINT; // Reduce existing zone by this length [mm]
	mShiftFrontEdge			: BOOL; // Shift front edge for reduction
END_VAR
VAR
	mIdx					: UINT; // Loop iterator
	mWindowIndex			: UINT; // Start window index
	mReductionWindowLength	: UINT; // Zone length in windows
	mReductionAllowed 		: BOOL; // Reduction valid
	mZoneEndWindowIndex		: UINT; // Zone end window index
	mZoneStartWindowIndex	: UINT; // Zone start window index
	mZoneEndPositionNew		: UDINT; // Zone end position after reduction
	mZoneStartPositionNew	: UDINT; // Zone start position after enlargement
END_VAR
VAR_INST
	OldZoneData				: ST_WindowTrackingZone; // Old tracking zone data
END_VAR
M_ShortenZone := FALSE;

// Validate inputs
IF mZoneIndex <= 0 OR
   mZoneIndex > MAX_NUMBER_OF_ZONES OR
   WindowSize = 0 THEN
   RETURN;
END_IF

IF ZoneTable[mZoneIndex].TU_Present THEN
	IF NOT mShiftFrontEdge THEN
		// Calculate new zone end position
		IF mReductionLength > ZoneTable[mZoneIndex].ZoneEndPosition THEN
			mZoneEndPositionNew := ZoneTable[mZoneIndex].ZoneEndPosition - mReductionLength + TotalTrackingLength;
			mReductionWindowLength := M_GetWindowIndex(M_GetAbsolutePosition(ZoneTable[mZoneIndex].ZoneEndPosition)) - M_GetWindowIndex(M_GetAbsolutePosition(mZoneEndPositionNew)) + MaxWindowIndex + 1;
		ELSE
			mZoneEndPositionNew := ZoneTable[mZoneIndex].ZoneEndPosition - mReductionLength;
			mReductionWindowLength := M_GetWindowIndex(M_GetAbsolutePosition(ZoneTable[mZoneIndex].ZoneEndPosition)) - M_GetWindowIndex(M_GetAbsolutePosition(mZoneEndPositionNew)) + 1;
		END_IF
		
		mWindowIndex := ZoneTable[mZoneIndex].ZoneEndWindowIndex;
		mReductionAllowed := TRUE;
		
		// Ensure reduction is possible
		FOR mIdx := 1 TO mReductionWindowLength DO
			// Is intended window index not occupied by TU
			IF WindowTable[mWindowIndex].State <> E_WindowTrackingWindowState.RESERVED THEN
				mReductionAllowed := FALSE;
				// Error
				fbDebugMsg.M_SendErrorMsg('M_ShortenZone - Reduction not possible, TU already in range of reduction.');	
				RETURN;
			END_IF
			
			mWindowIndex := mWindowIndex - 1;
			
			// Correct border overflow
			IF mWindowIndex = 0 THEN
				mWindowIndex := MaxWindowIndex;
			END_IF
		END_FOR
	ELSE
		// Calculate new zone start position
		IF ZoneTable[mZoneIndex].ZoneStartPosition + mReductionLength > TotalTrackingLength THEN
			mZoneStartPositionNew := ZoneTable[mZoneIndex].ZoneStartPosition + mReductionLength - TotalTrackingLength;
			mReductionWindowLength := M_GetWindowIndex(M_GetAbsolutePosition(mZoneStartPositionNew)) - M_GetWindowIndex(M_GetAbsolutePosition(ZoneTable[mZoneIndex].ZoneStartPosition)) + MaxWindowIndex + 1;
		ELSE
			mZoneStartPositionNew := ZoneTable[mZoneIndex].ZoneStartPosition + mReductionLength;
			mReductionWindowLength := M_GetWindowIndex(M_GetAbsolutePosition(mZoneStartPositionNew)) - M_GetWindowIndex(M_GetAbsolutePosition(ZoneTable[mZoneIndex].ZoneStartPosition)) + 1;
		END_IF
		
		mWindowIndex := ZoneTable[mZoneIndex].ZoneStartWindowIndex;
		mReductionAllowed := TRUE;
		
		// Ensure reduction is possible
		FOR mIdx := 1 TO mReductionWindowLength DO
			// Is intended window index not occupied by TU
			IF WindowTable[mWindowIndex].State <> E_WindowTrackingWindowState.RESERVED THEN
				mReductionAllowed := FALSE;
				// Error
				fbDebugMsg.M_SendErrorMsg('M_ShortenZone - Reduction not possible, TU already in range of reduction.');	
				RETURN;
			END_IF
			
			mWindowIndex := mWindowIndex + 1;
			
			// Correct border overflow
			IF mWindowIndex > MaxWindowIndex THEN
				mWindowIndex := mWindowIndex - MaxWindowIndex;
			END_IF
		END_FOR
	END_IF
END_IF

// When reduction is possible to be executed
IF mReductionAllowed THEN
	OldZoneData := ZoneTable[mZoneIndex];
	
	IF NOT mShiftFrontEdge THEN
		mWindowIndex := ZoneTable[mZoneIndex].ZoneEndWindowIndex;
	
		// Loop through all windows and assign new zone
		// Init
		mZoneEndWindowIndex := mWindowIndex;
		
		FOR mIdx := 1 TO mReductionWindowLength DO
			// Clear window
			MEMSET(ADR(WindowTable[mWindowIndex]), 0, SIZEOF(WindowTable[mWindowIndex]));
			
			mWindowIndex := mWindowIndex - 1;
			
			// Correct border overflow
			IF mWindowIndex = 0 THEN
				mWindowIndex := MaxWindowIndex;
			END_IF
				
			mZoneEndWindowIndex := mWindowIndex;
		END_FOR	
		
		// Update zone table
		ZoneTable[mZoneIndex].ZoneEndWindowIndex := mZoneEndWindowIndex;
		ZoneTable[mZoneIndex].ZoneEndPosition := mZoneEndPositionNew;
		ZoneTable[mZoneIndex].ZoneLength := ZoneTable[mZoneIndex].ZoneLength - mReductionLength;
		
		// Inform listener
		IF iEventListener <> 0 THEN
			iEventListener.M_TrackingZoneShortenedEvent(
				mTrackingZoneIndex 		:= mZoneIndex,
                mOldTrackingZoneData 	:= OldZoneData,
                mNewTrackingZoneDAta 	:= ZoneTable[mZoneIndex]);
		END_IF

		M_ShortenZone := TRUE;
	ELSE
		mWindowIndex := ZoneTable[mZoneIndex].ZoneStartWindowIndex;
	
		// Loop through all windows and assign new zone
		// Init
		mZoneStartWindowIndex := mWindowIndex;
		
		FOR mIdx := 1 TO mReductionWindowLength DO
			// Clear window
			MEMSET(ADR(WindowTable[mWindowIndex]), 0, SIZEOF(WindowTable[mWindowIndex]));
			
			mWindowIndex := mWindowIndex + 1;
			
			// Correct border overflow
			IF mWindowIndex > MaxWindowIndex THEN
				mWindowIndex := mWindowIndex - MaxWindowIndex;
			END_IF
				
			mZoneStartWindowIndex := mWindowIndex;
		END_FOR	
		
		// Update zone table
		ZoneTable[mZoneIndex].ZoneStartWindowIndex := mZoneStartWindowIndex;
		ZoneTable[mZoneIndex].ZoneStartPosition := mZoneStartPositionNew;
		ZoneTable[mZoneIndex].ZoneLength := ZoneTable[mZoneIndex].ZoneLength - mReductionLength;
		
		// Inform listener
		IF iEventListener <> 0 THEN
			iEventListener.M_TrackingZoneShortenedEvent(
				mTrackingZoneIndex 		:= mZoneIndex,
                mOldTrackingZoneData 	:= OldZoneData,
                mNewTrackingZoneDAta 	:= ZoneTable[mZoneIndex]);
		END_IF
		
		M_ShortenZone := TRUE;
	END_IF
END_IF
END_METHOD

/// Shortes a zone from window to its boder where no TU is in between
METHOD PROTECTED M_ShortenZoneAtWindow : BOOL // Returns true if successful, otherwise false
VAR_INPUT
	mZoneIndex			: UINT;
	mWindowIndex		: UINT; // Start window index
END_VAR
VAR_INST
	ShortenAfterTU 		: BOOL; // Shorten on side between zone end and tu end
	ShortenInFrontOfTU 	: BOOL; // Shorten on side between tu start and zone start
	ShortenLengthMM		: UINT; // Length to shorten
END_VAR
M_ShortenZoneAtWindow := FALSE;
ShortenAfterTU:= FALSE;
ShortenInFrontOfTU := FALSE;
ShortenLengthMM := 0;

// Validate inputs
IF mWindowIndex = 0 OR
   mWindowIndex > WindowTracking.MAX_NUMBER_OF_WINDOWS OR 
   mZoneIndex = 0 THEN
	RETURN;
END_IF
 
IF WindowTable[mWindowIndex].ZoneIndex <> mZoneIndex THEN
	RETURN;
END_IF

IF ZoneTable[mZoneIndex].TU_Present THEN
	// Find related border (No TU between window index and border)
	//        |
	//        v     TU
	//            ||||||
	//   |--------||||||----|
	//   

	// Check for no overflow between zone end and tu rear edge
	IF ZoneTable[mZoneIndex].ZoneEndWindowIndex >= ZoneTable[mZoneIndex].TU_EndWindowIndex THEN
		// Check if window index is between
		IF mWindowIndex >= ZoneTable[mZoneIndex].TU_EndWindowIndex AND
		   mWindowIndex <= ZoneTable[mZoneIndex].ZoneEndWindowIndex THEN
		   // Window for shorten found
		   ShortenAfterTU := TRUE;
		   ShortenLengthMM := UDINT_TO_UINT(ZoneTable[mZoneIndex].ZoneEndPosition - ((mWindowIndex-1) * WindowSize));
		END_IF
	ELSE
		// Check if window index is between
		IF mWindowIndex >= ZoneTable[mZoneIndex].TU_EndWindowIndex THEN
		   	// Window for shorten found
		  	ShortenAfterTU := TRUE;
		   	ShortenLengthMM := UDINT_TO_UINT(ZoneTable[mZoneIndex].ZoneEndPosition + TotalTrackingLength - ((mWindowIndex-1) * WindowSize));
			
		ELSIF mWindowIndex <= ZoneTable[mZoneIndex].ZoneEndWindowIndex THEN
			// Window for shorten found
		   	ShortenAfterTU := TRUE;
		   	ShortenLengthMM := UDINT_TO_UINT(ZoneTable[mZoneIndex].ZoneEndPosition - ((mWindowIndex-1) * WindowSize));	
		END_IF
	END_IF
	
	// Check for no overflow between zone end and tu rear edge
	IF ZoneTable[mZoneIndex].TU_StartWindowIndex >= ZoneTable[mZoneIndex].ZoneStartWindowIndex THEN
		// Check if window index is between
		IF mWindowIndex >= ZoneTable[mZoneIndex].ZoneStartWindowIndex AND
		   mWindowIndex <= ZoneTable[mZoneIndex].TU_StartWindowIndex THEN
		   // Window for shorten found
		   ShortenInFrontOfTU := TRUE;
		   ShortenLengthMM := UDINT_TO_UINT((mWindowIndex * WindowSize) - ZoneTable[mZoneIndex].ZoneStartPosition);
		END_IF
	ELSE
		// Check if window index is between
		IF mWindowIndex >= ZoneTable[mZoneIndex].ZoneStartWindowIndex THEN
		   	// Window for shorten found
		   	ShortenInFrontOfTU := TRUE;
		   	ShortenLengthMM := UDINT_TO_UINT((mWindowIndex * WindowSize) - ZoneTable[mZoneIndex].ZoneStartPosition);
		   
		ELSIF mWindowIndex <= ZoneTable[mZoneIndex].TU_StartWindowIndex THEN
			// Window for shorten found
		   	ShortenInFrontOfTU := TRUE;
		   	ShortenLengthMM := UDINT_TO_UINT((mWindowIndex * WindowSize) + TotalTrackingLength - ZoneTable[mZoneIndex].ZoneStartPosition);
		END_IF
	END_IF

	// When window was found inside a valid area of the zone
	IF ShortenInFrontOfTU OR ShortenAfterTU THEN
		IF ShortenInFrontOfTU THEN
			M_ShortenZoneAtWindow := M_ShortenZone(mZoneIndex, ShortenLengthMM, TRUE);
	  	ELSE
			M_ShortenZoneAtWindow := M_ShortenZone(mZoneIndex, ShortenLengthMM, FALSE);
		END_IF
	END_IF
END_IF
END_METHOD

/// All Zones get deleted if they completly (Rear edge) left TrackingLength
/// Default: Enabled
PROPERTY P_DeleteZoneTrackingEnd : BOOL // Returns true if enabled, otherwise false
GET
P_DeleteZoneTrackingEnd := DeleteZoneTrackingEnd;
END_GET
SET
DeleteZoneTrackingEnd := P_DeleteZoneTrackingEnd;
END_SET
END_PROPERTY

/// Additional tracking length. Can be used to allow more additional space for reservations.
PROPERTY P_TrackingAddition : UDINT // Additional tracking distance
GET
P_TrackingAddition := TrackingAddition;
END_GET
SET
TrackingAddition := P_TrackingAddition;
END_SET
END_PROPERTY

/// Access to Ongoing trasfer list  for read operations
/// Remark: User has to ensure that writing does not influence the process in a bad way.
{attribute 'suppress_wrn_C0410'}
PROPERTY P_TransferList : REFERENCE TO ARRAY[1..TRANSFER_TABLE_SIZE] OF ST_WindowTrackingTransfer
GET
P_TransferList REF= OngoingTransferList;
END_GET
END_PROPERTY

/// Returns currently available amount of TUs
PROPERTY P_TU_Count : INT
GET
P_TU_Count := TU_Count;
END_GET
END_PROPERTY

/// Access to Window table  for read operations
/// Remark: User has to ensure that writing does not influence the process in a bad way.
{attribute 'suppress_wrn_C0410'}
PROPERTY P_WindowTable : REFERENCE TO ARRAY[1..WindowTracking.MAX_NUMBER_OF_WINDOWS] OF ST_WindowTrackingWindow;
GET
P_WindowTable REF= WindowTable;
END_GET
END_PROPERTY

/// Returns currently available amount of Zones
PROPERTY P_ZoneCount : INT
GET
P_ZoneCount := ZoneCount;
END_GET
END_PROPERTY

/// Access to Zone table  for read operations
/// Remark: User has to ensure that writing does not influence the process in a bad way.
{attribute 'suppress_wrn_C0410'}
PROPERTY P_ZoneTable : REFERENCE TO ARRAY[1..WindowTracking.MAX_NUMBER_OF_ZONES] OF ST_WindowTrackingZone;
GET
P_ZoneTable REF= ZoneTable;
END_GET
END_PROPERTY

END_FUNCTION_BLOCK

(* stored: Version 1.1.0.1, ProductVersion 3.1.4024.4
   POU FB_WindowTracking: Id {587d5bf3-e64f-4583-bce1-15727290ddd2}, SpecialFunc None
   Method M_AddTU: Id {cde32322-776f-4203-9221-f32669cbbba5}
   Method M_AddTU_FE: Id {60b231e4-640a-4b56-b940-2b211cb1d291}
   Method M_AddTU_RE: Id {d814d3c2-4ca0-4441-97f9-54672d98a6e9}
   Method M_AddZoneToPTL: Id {029071cc-66ac-4eb5-8079-f6c131fc43de}
   Method M_AdjustFE: Id {90ac2b5f-1a03-4f0b-b7ec-03fd6714b6f4}
   Method M_AdjustRE: Id {b8803c21-0d1d-470d-9b12-1b36daff3674}
   Method M_AllocateFixedZone: Id {1449a464-e5d4-49bd-a669-1b641b28291e}
   Method M_AllocateNextFreeZone: Id {eab9f650-b68c-4bde-842a-abec02129d7e}
   Method M_AssignNextFreeZone: Id {7a98cebf-1bd0-48b7-8336-0cab1fb97179}
   Method M_CalculateTotalTrackingLength: Id {144ec777-0eb0-4a17-8a02-53eb336cb8ca}
   Method M_ClearTables: Id {93e3ebd3-49ec-4edc-8e35-8aa72f839642}
   Method M_ClearWindow: Id {f2025eb8-c615-4476-9dfa-fd43c0d6fbe2}
   Method M_DeleteZone: Id {5220ccb4-4fa0-48d6-a82d-9481c1a12da1}
   Method M_EnlargeZone: Id {c49b1261-8958-4b76-beec-b7d48a56b3f7}
   Method M_FlushDistance: Id {9d553746-93ac-4eb4-86cd-df210fe81771}
   Method M_GetAbsolutePosition: Id {128fd462-103b-46d2-b1da-feef9d46088f}
   Method M_GetDistanceToTU_End: Id {dddf1dcf-3adf-4d1f-a800-63fca8c7a466}
   Method M_GetDistanceToTU_Start: Id {59b019ca-0cb9-48d4-bb7b-66b7d0cab66b}
   Method M_GetDistanceToZoneEnd: Id {2733d983-dc18-42dc-a3b0-91be96617f09}
   Method M_GetDistanceToZoneStart: Id {e8fcc9a7-abdd-4e09-ba21-88371a6dc389}
   Method M_GetFirstZoneIndex: Id {e5e4973c-2e72-445e-8ad4-e263073a3f35}
   Method M_GetLastZoneIndex: Id {3226c821-2878-49c4-89bd-6e7e6a3b3a33}
   Method M_GetPendingAssignments: Id {a85c7b51-02a3-4bd6-bc9a-d5e2d24a16e8}
   Method M_GetTrackingPosition: Id {451239b8-aecc-4af8-8dcd-79ac997b0c57}
   Method M_GetTU_EndPosition: Id {5069c6a2-a844-47af-bbcc-81246e106620}
   Method M_GetTU_StartPosition: Id {8035e856-6be3-441a-b14c-2028d644d3c8}
   Method M_GetWindowIndex: Id {db807389-4f66-4298-9fcc-481d457369df}
   Method M_GetZoneEndPosition: Id {ab871644-5af0-4f5b-a7e8-1e55b88d127a}
   Method M_GetZoneIndex: Id {e7409bb3-72bd-4e6d-9217-37f942d4a3bb}
   Method M_GetZoneStartPosition: Id {23a80f7e-32e9-48d6-b83e-a5e9a1e01229}
   Method M_InhibitShifting: Id {26a226be-b2de-4cf9-b49b-40059a703657}
   Method M_Init: Id {31e6e445-2730-4f9c-9aab-9f9a8eda721c}
   Method M_InsertNewZoneIndex: Id {948b1b40-460d-43fd-a302-f458265185cb}
   Method M_IsShiftable: Id {7beaad1c-246f-428e-8dbe-ae6759d8f438}
   Method M_IsTU_InRange: Id {f9283e40-2538-4614-9dcf-907e141bb5fb}
   Method M_IsTU_Present: Id {b714aff5-1e37-4620-96ee-24635cd48a86}
   Method M_IsZoneInRange: Id {07774e1c-639f-4c8c-b110-4045bb303043}
   Method M_MakeSpace: Id {2fd2b491-b214-4398-855b-581cc663a1fa}
   Method M_MakeSpaceByWindows: Id {36390a8b-f894-42fb-9c3f-9b4a196075e7}
   Method M_ManageOngoingTransfers: Id {8207db95-1288-4ff9-9f2d-82b7de88802b}
   Method M_MonitorZonesPTL: Id {2396352b-4deb-4781-bc82-8822c1c85676}
   Method M_MoveZone: Id {ddc345d4-ce37-4962-8074-84103112b9d9}
   Method M_MoveZoneFE: Id {673d8e4e-a51f-4c1d-b999-0cc4b7b68e7b}
   Method M_MoveZoneRE: Id {d8d325ed-3e2d-46c7-b7bf-52757b03c146}
   Method M_RemoveZoneFromPTL: Id {00a5ee10-279d-49ae-874b-0754242c2380}
   Method M_RemoveZoneFromTransferList: Id {fe181709-b97e-4ebe-b879-7535ed1860ba}
   Method M_ReserveZone: Id {cb55d34d-3ca6-471c-a0a1-dc936395962b}
   Method M_ResyncOnlyFE: Id {84a25842-3cdc-4730-ab3c-c506689a1078}
   Method M_ResyncOnlyRE: Id {6fdf8443-35ff-417f-999c-f1d4a06c3d53}
   Method M_ResyncTU_FE: Id {0632ccab-4dcd-4b74-80ce-38bc20c7e61d}
   Method M_ResyncTU_RE: Id {67633d5e-db15-4da9-a88d-8ddb1e0e7b93}
   Method M_ShiftZone: Id {08440ea1-4b89-4401-a375-e1711cabebf6}
   Method M_ShortenZone: Id {b360cdc1-2dbe-47ee-b030-dd6656ea1fa6}
   Method M_ShortenZoneAtWindow: Id {40bc74b9-efaf-443d-a546-1a2effa19b65}
   Property P_DeleteZoneTrackingEnd: Id {05b77ade-6117-4d16-b592-a6a32a63f0f8}
   Get Get: Id {b3dbf710-efe8-4525-9cda-2cd13af61e10}
   Set Set: Id {7339db5b-264c-45b0-8047-38de9149b495}
   Property P_TrackingAddition: Id {103e273b-67e9-4be0-9ba7-cc481966cdea}
   Get Get: Id {f07fbaf0-494c-46da-bd86-5c4d5f4a7c99}
   Set Set: Id {02a9110a-1f66-4b4a-a9e4-4390c31a087a}
   Property P_TransferList: Id {80d5faef-a0d4-42b3-8525-5781194f7b0e}
   Get Get: Id {2c3a2542-cf5c-4e86-bd14-1b1952f29c80}
   Property P_TU_Count: Id {6b488f27-acf7-47b0-b092-606d3d96af85}
   Get Get: Id {a2dbed7c-8df2-45d1-beda-599b3c7eef34}
   Property P_WindowTable: Id {2e36c3fe-c255-45dc-bcd3-e00da9932bce}
   Get Get: Id {ce938b07-cb0d-448b-9e12-2593cb3b8350}
   Property P_ZoneCount: Id {8a29b4a6-8470-4188-bb5d-98cb614f5c8a}
   Get Get: Id {2cc354f9-c67a-4891-ae45-61c8349df8bf}
   Property P_ZoneTable: Id {728e378f-0db2-4831-b262-bd53ec917f5b}
   Get Get: Id {e5840375-a011-44eb-9f62-c42ae7510d84} *)
